ACTION A_LeftTopMove:
IF LeftTopMove THEN
LeftTopBusy:=TRUE;
LeftTopDone:=FALSE;
fb_ton_debug_1(PT:=t#10s);
(*×îºóÔÙ¼ì²éÒ»±éñîºÏ£¬²»ñîºÏÎªÕýÈ·×´Ì¬*)
IF LeftTopLin.NcToPlc.CoupleState<>0 OR LeftBottomLin.NcToPlc.CoupleState<>0
			OR RightTopLin.NcToPlc.CoupleState<>0 OR RightBottomLin.NcToPlc.CoupleState<>0 THEN
			ErrorID:=1;
			LeftTopState:=-100;
END_IF
A_MoveMC();
CASE LeftTopState OF
	0:
		IF Top_MC_MoveAbsolute.Error OR Bottom_MC_MoveAbsolute.Error
			OR RightTopLin_MC_MoveAbsolute.Error OR RightBottomLin_MC_MoveAbsolute.Error THEN		(*¼ì²éMC Error*)
			ErrorID:=2;
			LeftTopState:=99;
		ELSIF leftTopLin.Status.NotMoving AND  leftBottomLin.Status.NotMoving
			 AND RightTopLin.Status.NotMoving AND RightBottomLin.Status.NotMoving THEN	(*Öá¶¼´¦ÓÚÍ£Ö¹×´Ì¬Ê±£¬×ªÏÂÒ»²½*)
			LeftTopState:=1;
		END_IF
	1:
		Top_MC_MoveAbsolute.Position:=LeftTopPosition;
		Top_MC_MoveAbsolute.Velocity:=LeftTopVelocity;
		Top_MC_MoveAbsolute.Execute:=TRUE;
		fb_ton_debug_1.IN:=TRUE;
		LeftTopState:=2;
	2:
		IF RightTopLin.Status.Moving OR LeftBottomLin.Status.Moving OR RightBottomLin.Status.Moving THEN	(*³ýÁËÔË¶¯Öá¶¯£¬ÆäÓàÖáÓÐ¶¯£¬´íÎó*)
			ErrorID:=3;
			LeftTopState:=-100;
		ELSIF NOT Top_MC_MoveAbsolute.Done THEN		(*ÔË¶¯ÖÐ£¬¼ì²éDoneÐÅºÅ£¬Ã»ÓÐÔòÑ­»·£¬³¬Ê±±¨´í*)
			(*IF NOT  fb_ton.Q THEN
				LeftTopState:=2;
			ELSE
				ErrorID:=5;
				LeftTopState:=-100;
			END_IF*)
			LeftTopState:=2;
		ELSIF Top_MC_MoveAbsolute.Done THEN		(*ÔË¶¯Íê³É£¬×ªÏÂÒ»²½*)
				LeftTopState:=88;
		END_IF
		(*½ÓÊÕµ½stopÐÅºÅÊ±£¬reset×´Ì¬*)
		IF LeftTopReset THEN
			LeftTopState:=89;
		END_IF

	88:
		LeftTopMove:=FALSE;
		LeftTopState:=0;
		LeftTopBusy:=FALSE;
		LeftTopDone:=TRUE;
		Error:=FALSE;
		ErrorID:=0;
		Top_MC_MoveAbsolute.Execute:=FALSE;
		fb_ton_debug_1.IN:=FALSE;
	89:
		LeftTopMove:=FALSE;
		LeftTopState:=0;
		LeftTopBusy:=FALSE;
		LeftTopDone:=FALSE;
		Error:=FALSE;
		ErrorID:=0;
		Top_MC_MoveAbsolute.Execute:=FALSE;
		fb_ton_debug_1.IN:=FALSE;
	99:
		LeftTopMove:=FALSE;
		LeftTopState:=99;
		LeftTopBusy:=FALSE;
		LeftTopDone:=FALSE;
		Error:=TRUE;
		Top_MC_MoveAbsolute.Execute:=FALSE;
		fb_ton_debug_1.IN:=FALSE;
	-100:
		FB_PlcEmergencyStop();
		LeftTopMove:=FALSE;
		LeftTopState:=-100;
		LeftTopBusy:=FALSE;
		LeftTopDone:=FALSE;
		Error:=TRUE;
		Top_MC_MoveAbsolute.Execute:=FALSE;
		fb_ton_debug_1.IN:=FALSE;
END_CASE
END_IF
END_ACTION

ACTION A_MoveMC:
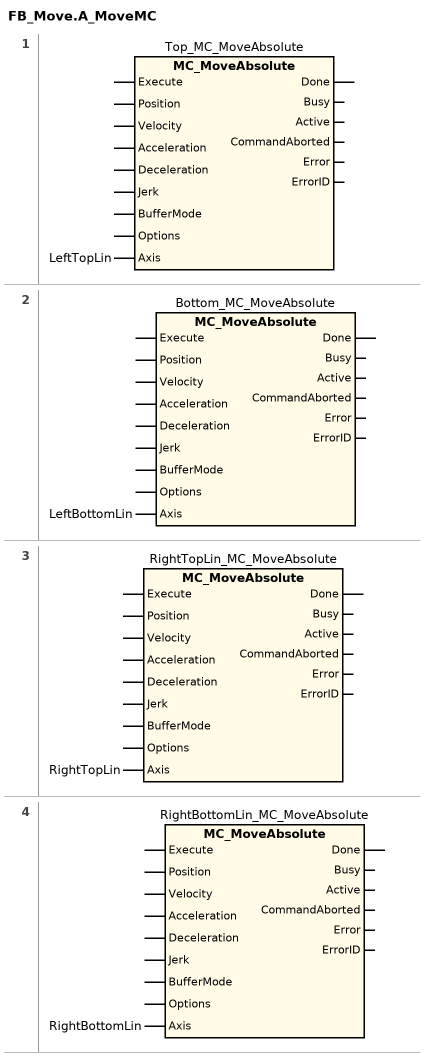
// NETWORK 1
Top_MC_MoveAbsolute(Axis := LeftTopLin); // MC_MoveAbsolute

// NETWORK 2
Bottom_MC_MoveAbsolute(Axis := LeftBottomLin); // MC_MoveAbsolute

// NETWORK 3
RightTopLin_MC_MoveAbsolute(Axis := RightTopLin); // MC_MoveAbsolute

// NETWORK 4
RightBottomLin_MC_MoveAbsolute(Axis := RightBottomLin); // MC_MoveAbsolute
END_ACTION

ACTION A_RightBottomMove:
IF RightBottomMove THEN
RightBottomBusy:=TRUE;
RightBottomDone:=FALSE;
fb_ton_debug_4(PT:=t#10s);
(*×îºóÔÙ¼ì²éÒ»±éñîºÏ£¬²»ñîºÏÎªÕýÈ·×´Ì¬*)
IF LeftTopLin.NcToPlc.CoupleState<>0 OR LeftBottomLin.NcToPlc.CoupleState<>0
			OR RightTopLin.NcToPlc.CoupleState<>0 OR RightBottomLin.NcToPlc.CoupleState<>0 THEN
			ErrorID:=1;
			RightBottomState:=-100;
END_IF
A_MoveMC();
CASE RightBottomState OF
	0:
		IF Top_MC_MoveAbsolute.Error OR Bottom_MC_MoveAbsolute.Error
			OR RightTopLin_MC_MoveAbsolute.Error OR RightBottomLin_MC_MoveAbsolute.Error THEN		(*¼ì²éMC Error*)
			ErrorID:=2;
			RightBottomState:=99;
		ELSIF leftTopLin.Status.NotMoving AND  leftBottomLin.Status.NotMoving
			 AND RightTopLin.Status.NotMoving AND RightBottomLin.Status.NotMoving THEN	(*Öá¶¼´¦ÓÚÍ£Ö¹×´Ì¬Ê±£¬×ªÏÂÒ»²½*)
			RightBottomState:=1;
		END_IF
	1:
		RightBottomLin_MC_MoveAbsolute.Position:=RightBottomPosition;
		RightBottomLin_MC_MoveAbsolute.Velocity:=RightBottomVelocity;
		RightBottomLin_MC_MoveAbsolute.Execute:=TRUE;
		fb_ton_debug_4.IN:=TRUE;
		RightBottomState:=2;
	2:
		IF LeftTopLin.Status.Moving OR RightTopLin.Status.Moving  OR LeftBottomLin.Status.Moving THEN	(*³ýÁËÔË¶¯Öá¶¯£¬ÆäÓàÖáÓÐ¶¯£¬´íÎó*)
			ErrorID:=3;
			RightBottomState:=-100;
		ELSIF NOT RightBottomLin_MC_MoveAbsolute.Done THEN		(*ÔË¶¯ÖÐ£¬¼ì²éDoneÐÅºÅ£¬Ã»ÓÐÔòÑ­»·£¬³¬Ê±±¨´í*)
			(*IF NOT  fb_ton.Q THEN
				LeftTopState:=2;
			ELSE
				ErrorID:=5;
				LeftTopState:=-100;
			END_IF*)
			RightBottomState:=2;
		ELSIF RightBottomLin_MC_MoveAbsolute.Done THEN		(*ÔË¶¯Íê³É£¬×ªÏÂÒ»²½*)
				RightBottomState:=88;
		END_IF
		(*½ÓÊÕµ½stopÐÅºÅÊ±£¬reset×´Ì¬*)
		IF RightBottomReset THEN
			RightBottomState:=89;
		END_IF

	88:
		RightBottomMove:=FALSE;
		RightBottomState:=0;
		RightBottomBusy:=FALSE;
		RightBottomDone:=TRUE;
		Error:=FALSE;
		ErrorID:=0;
		RightBottomLin_MC_MoveAbsolute.Execute:=FALSE;
		fb_ton_debug_4.IN:=FALSE;
	89:
		RightBottomMove:=FALSE;
		RightBottomState:=0;
		RightBottomBusy:=FALSE;
		RightBottomDone:=FALSE;
		Error:=FALSE;
		ErrorID:=0;
		RightBottomLin_MC_MoveAbsolute.Execute:=FALSE;
		fb_ton_debug_4.IN:=FALSE;
	99:
		RightBottomMove:=FALSE;
		RightBottomState:=99;
		RightBottomBusy:=FALSE;
		RightBottomDone:=FALSE;
		Error:=TRUE;
		RightBottomLin_MC_MoveAbsolute.Execute:=FALSE;
		fb_ton_debug_4.IN:=FALSE;
	-100:
		FB_PlcEmergencyStop();
		RightBottomMove:=FALSE;
		RightBottomState:=-100;
		RightBottomBusy:=FALSE;
		RightBottomDone:=FALSE;
		Error:=TRUE;
		RightBottomLin_MC_MoveAbsolute.Execute:=FALSE;
		fb_ton_debug_4.IN:=FALSE;
END_CASE
END_IF
END_ACTION

ACTION A_RightTopMove:
IF RightTopMove THEN
RightTopBusy:=TRUE;
RightTopDone:=FALSE;
fb_ton_debug_2(PT:=t#10s);
(*×îºóÔÙ¼ì²éÒ»±éñîºÏ£¬²»ñîºÏÎªÕýÈ·×´Ì¬*)
IF LeftTopLin.NcToPlc.CoupleState<>0 OR LeftBottomLin.NcToPlc.CoupleState<>0
			OR RightTopLin.NcToPlc.CoupleState<>0 OR RightBottomLin.NcToPlc.CoupleState<>0 THEN
			ErrorID:=1;
			RightTopState:=-100;
END_IF
A_MoveMC();
CASE RightTopState OF
	0:
		IF Top_MC_MoveAbsolute.Error OR Bottom_MC_MoveAbsolute.Error
			OR RightTopLin_MC_MoveAbsolute.Error OR RightBottomLin_MC_MoveAbsolute.Error THEN		(*¼ì²éMC Error*)
			ErrorID:=2;
			RightTopState:=99;
		ELSIF leftTopLin.Status.NotMoving AND  leftBottomLin.Status.NotMoving
			 AND RightTopLin.Status.NotMoving AND RightBottomLin.Status.NotMoving THEN	(*Öá¶¼´¦ÓÚÍ£Ö¹×´Ì¬Ê±£¬×ªÏÂÒ»²½*)
			RightTopState:=1;
		END_IF
	1:
		RightTopLin_MC_MoveAbsolute.Position:=RightTopPosition;
		RightTopLin_MC_MoveAbsolute.Velocity:=RightTopVelocity;
		RightTopLin_MC_MoveAbsolute.Execute:=TRUE;
		fb_ton_debug_2.IN:=TRUE;
		RightTopState:=2;
	2:
		IF LeftTopLin.Status.Moving OR LeftBottomLin.Status.Moving OR RightBottomLin.Status.Moving THEN	(*³ýÁËÔË¶¯Öá¶¯£¬ÆäÓàÖáÓÐ¶¯£¬´íÎó*)
			ErrorID:=3;
			RightTopState:=-100;
		ELSIF NOT RightTopLin_MC_MoveAbsolute.Done THEN		(*ÔË¶¯ÖÐ£¬¼ì²éDoneÐÅºÅ£¬Ã»ÓÐÔòÑ­»·£¬³¬Ê±±¨´í*)
			(*IF NOT  fb_ton.Q THEN
				LeftTopState:=2;
			ELSE
				ErrorID:=5;
				LeftTopState:=-100;
			END_IF*)
			RightTopState:=2;
		ELSIF RightTopLin_MC_MoveAbsolute.Done THEN		(*ÔË¶¯Íê³É£¬×ªÏÂÒ»²½*)
				RightTopState:=88;
		END_IF
		(*½ÓÊÕµ½stopÐÅºÅÊ±£¬reset×´Ì¬*)
		IF RightTopReset THEN
			RightTopState:=89;
		END_IF

	88:
		RightTopMove:=FALSE;
		RightTopState:=0;
		RightTopBusy:=FALSE;
		RightTopDone:=TRUE;
		Error:=FALSE;
		ErrorID:=0;
		RightTopLin_MC_MoveAbsolute.Execute:=FALSE;
		fb_ton_debug_2.IN:=FALSE;
	89:
		RightTopMove:=FALSE;
		RightTopState:=0;
		RightTopBusy:=FALSE;
		RightTopDone:=FALSE;
		Error:=FALSE;
		ErrorID:=0;
		RightTopLin_MC_MoveAbsolute.Execute:=FALSE;
		fb_ton_debug_2.IN:=FALSE;
	99:
		RightTopMove:=FALSE;
		RightTopState:=99;
		RightTopBusy:=FALSE;
		RightTopDone:=FALSE;
		Error:=TRUE;
		RightTopLin_MC_MoveAbsolute.Execute:=FALSE;
		fb_ton_debug_2.IN:=FALSE;
	-100:
		FB_PlcEmergencyStop();
		RightTopMove:=FALSE;
		RightTopState:=-100;
		RightTopBusy:=FALSE;
		RightTopDone:=FALSE;
		Error:=TRUE;
		RightTopLin_MC_MoveAbsolute.Execute:=FALSE;
		fb_ton_debug_2.IN:=FALSE;
END_CASE
END_IF
END_ACTION

ACTION A_TaperMove:
IF TaperMove THEN
TaperBusy:=TRUE;
TaperDone:=FALSE;
fb_ton(PT:=t#80s);
(*×îºóÔÙ¼ì²éÒ»±éñîºÏ£¬²»ñîºÏÎªÕýÈ·×´Ì¬*)
IF LeftTopLin.NcToPlc.CoupleState<>0 OR LeftBottomLin.NcToPlc.CoupleState<>0
			OR RightTopLin.NcToPlc.CoupleState<>0 OR RightBottomLin.NcToPlc.CoupleState<>0 THEN
			ErrorID:=1;
			TaperState:=-100;
END_IF
(*×ó²àÉÏÏÂÖá¶¯£¬ESTOP*)
IF LeftTopLin.Status.Moving OR LeftBottomLin.Status.Moving THEN
			ErrorID:=2;
			TaperState:=-100;
END_IF
(*ÓÒÉÏ¶¯¡¢ÓÒÏÂ²»¶¯£¬»òÕßÓÒÏÂ¶¯¡¢ÓÒÉÏ²»¶¯¡£ESTOP*)
IF (RightTopLin.Status.Moving AND RightBottomLin.Status.NotMoving) OR (RightTopLin.Status.NotMoving AND RightBottomLin.Status.Moving) THEN
			ErrorID:=3;
			TaperState:=-100;
END_IF
A_MoveMC();
CASE TaperState OF

	0:
		IF RightTopLin.Status.Moving OR RightBottomLin.Status.Moving THEN	(*ÓÒ²àÉÏÏÂÖáÕýÔÚÔËÐÐ£¬Ñ­»·¸Ã²½µÈ´ý*)
			TaperState:=88;
		ELSIF Top_MC_MoveAbsolute.Error OR Bottom_MC_MoveAbsolute.Error THEN		(*¼ì²éMC Error*)
			ErrorID:=4;
			TaperState:=99;
		ELSIF leftTopLin.Status.NotMoving AND  leftBottomLin.Status.NotMoving
			 AND RightTopLin.Status.NotMoving AND RightBottomLin.Status.NotMoving THEN	(*Öá¶¼´¦ÓÚÍ£Ö¹×´Ì¬Ê±£¬×ªÏÂÒ»²½*)
			TaperState:=1;
		END_IF
	1:
		RightTopLin_MC_MoveAbsolute.Position:=TaperPosition;
		RightTopLin_MC_MoveAbsolute.Velocity:=TaperVelocity;
		RightBottomLin_MC_MoveAbsolute.Position:=TaperPosition;
		RightBottomLin_MC_MoveAbsolute.Velocity:=TaperVelocity;
		RightTopLin_MC_MoveAbsolute.Execute:=TRUE;
		RightBottomLin_MC_MoveAbsolute.Execute:=TRUE;
		fb_ton.IN:=TRUE;
		TaperState:=2;
	2:
		IF leftTopLin.Status.Moving OR   leftBottomLin.Status.Moving THEN		(*×ó²àÉÏÏÂÖá¶¯£¬ESTOP*)
			ErrorID:=5;
			TaperState:=-100;
		ELSIF  (RightTopLin.Status.Moving AND RightBottomLin.Status.NotMoving) OR (RightTopLin.Status.NotMoving AND RightBottomLin.Status.Moving) THEN
			ErrorID:=6;
			TaperState:=-100;
		ELSIF NOT RightTopLin_MC_MoveAbsolute.Done OR NOT  RightBottomLin_MC_MoveAbsolute.Done THEN		(*ÔË¶¯ÖÐ£¬¼ì²éDoneÐÅºÅ£¬Ã»ÓÐÔòÑ­»·£¬³¬Ê±±¨´í*)
			(*IF NOT  fb_ton.Q THEN
				TaperState:=2;
			ELSE
				ErrorID:=5;
				TaperState:=-100;
			END_IF*)
			TaperState:=2;
		ELSIF RightTopLin_MC_MoveAbsolute.Done  AND  RightBottomLin_MC_MoveAbsolute.Done THEN		(*ÔË¶¯Íê³É£¬×ªÏÂÒ»²½*)
				TaperState:=88;
		END_IF
		(*½ÓÊÕµ½stopÐÅºÅÊ±£¬reset×´Ì¬*)
		IF TaperReset THEN
			TaperState:=89;
		END_IF

	88:
		TaperMove:=FALSE;
		TaperState:=0;
		TaperBusy:=FALSE;
		TaperDone:=TRUE;
		Error:=FALSE;
		ErrorID:=0;
		RightTopLin_MC_MoveAbsolute.Execute:=FALSE;
		RightBottomLin_MC_MoveAbsolute.Execute:=FALSE;
		fb_ton.IN:=FALSE;
	89:
		TaperMove:=FALSE;
		TaperState:=0;
		TaperBusy:=FALSE;
		TaperDone:=FALSE;
		Error:=FALSE;
		ErrorID:=0;
		RightTopLin_MC_MoveAbsolute.Execute:=FALSE;
		RightBottomLin_MC_MoveAbsolute.Execute:=FALSE;
		fb_ton.IN:=FALSE;
	99:
		TaperMove:=FALSE;
		TaperState:=99;
		TaperBusy:=FALSE;
		TaperDone:=FALSE;
		Error:=TRUE;
		RightTopLin_MC_MoveAbsolute.Execute:=FALSE;
		RightBottomLin_MC_MoveAbsolute.Execute:=FALSE;
		fb_ton.IN:=FALSE;
	-100:
		FB_PlcEmergencyStop();
		TaperMove:=FALSE;
		TaperState:=-100;
		TaperBusy:=FALSE;
		TaperDone:=FALSE;
		Error:=TRUE;
		RightTopLin_MC_MoveAbsolute.Execute:=FALSE;
		RightBottomLin_MC_MoveAbsolute.Execute:=FALSE;
		fb_ton.IN:=FALSE;
END_CASE
END_IF
END_ACTION

ACTION A_TopMove:
IF TopMove THEN
TopBusy:=TRUE;
TopDone:=FALSE;
fb_ton1(PT:=t#80s);(*2mm/s max spees,120mmÐÐ³Ì£¬60sÄÚ×ßÍê*)
A_MoveMC();
CASE TopState OF
	0:
		IF Top_MC_MoveAbsolute.Error OR RightTopLin_MC_MoveAbsolute.Error THEN		(*¼ì²éMC Error*)
			ErrorID:=2;
			TopState:=99;
		END_IF
		TopState:=1;
	1:
		Top_MC_MoveAbsolute.Position:=TopPosition;
		Top_MC_MoveAbsolute.Velocity:=TopVelocity;
		Top_MC_MoveAbsolute.Execute:=TRUE;
		RightTopLin_MC_MoveAbsolute.Position:=TopPosition;
		RightTopLin_MC_MoveAbsolute.Velocity:=TopVelocity;
		RightTopLin_MC_MoveAbsolute.Execute:=TRUE;
		fb_ton1.IN:=TRUE;
		TopState:=2;
	2:
		IF leftBottomLin.Status.Moving OR RightBottomLin.Status.Moving THEN	(*ÏÂÁº¶¯,ESTOP*)
			ErrorID:=3;
			TopState:=-100;
		ELSIF  (LeftTopLin.Status.Moving AND  RightTopLin.Status.NotMoving)
				OR (RightTopLin.Status.Moving AND  LeftTopLin.Status.NotMoving) THEN			(*Ò»Öá¶¯£¬ÁíÒ»Öá²»¶¯£¬½ô¼±×´Ì¬*)
			ErrorID:=4;
			TopState:=-100;
		ELSIF NOT Top_MC_MoveAbsolute.Done OR NOT RightTopLin_MC_MoveAbsolute.Done THEN		(*ÔË¶¯ÖÐ£¬¼ì²éDoneÐÅºÅ£¬Ã»ÓÐÔòÑ­»·£¬³¬Ê±±¨´í*)
			TopState:=2;
		ELSIF Top_MC_MoveAbsolute.Done AND RightTopLin_MC_MoveAbsolute.Done THEN		(*ÔË¶¯Íê³É£¬×ªÏÂÒ»²½*)
				TopState:=88;
		END_IF
		(*½ÓÊÕµ½stopÐÅºÅÊ±£¬reset×´Ì¬*)
		IF TopReset THEN
			TopState:=89;
		END_IF

	88:
		TopMove:=FALSE;
		TopState:=0;
		TopBusy:=FALSE;
		TopDone:=TRUE;
		Error:=FALSE;
		ErrorID:=0;
		Top_MC_MoveAbsolute.Execute:=FALSE;
		RightTopLin_MC_MoveAbsolute.Execute:=FALSE;
		fb_ton1.IN:=FALSE;
	89:
		TopMove:=FALSE;
		TopState:=0;
		TopBusy:=FALSE;
		TopDone:=FALSE;
		Error:=FALSE;
		ErrorID:=0;
		Top_MC_MoveAbsolute.Execute:=FALSE;
		RightTopLin_MC_MoveAbsolute.Execute:=FALSE;
		fb_ton1.IN:=FALSE;
	99:
		TopMove:=FALSE;
		TopState:=99;
		TopBusy:=FALSE;
		TopDone:=FALSE;
		Error:=TRUE;
		Top_MC_MoveAbsolute.Execute:=FALSE;
		RightTopLin_MC_MoveAbsolute.Execute:=FALSE;
		fb_ton1.IN:=FALSE;
	-100:
		FB_PlcEmergencyStop();
		TopMove:=FALSE;
		TopState:=-100;
		TopBusy:=FALSE;
		TopDone:=FALSE;
		Error:=TRUE;
		Top_MC_MoveAbsolute.Execute:=FALSE;
		RightTopLin_MC_MoveAbsolute.Execute:=FALSE;
		fb_ton1.IN:=FALSE;
END_CASE
END_IF
END_ACTION

END_FUNCTION_BLOCK

// ---- POUs/CommonFB/MainFB/FB_Stop.TcPOU
FUNCTION_BLOCK FB_Stop
VAR_INPUT
(*È«¾Ö*)
	Mode:DINT;
	PowerState:BOOL;
	CoupleState:DINT;
	(*GapMode*)
	GapStop:BOOL;
	(*BCGapMode*)
	BCGapStop:BOOL;
	(*SingleCarrierMode*)
	TopStop:BOOL;
	BottomStop:BOOL;
	(*TaperMode*)
	TaperStop:BOOL;
	(*DebugMode*)
	LeftTopStop:BOOL;
	RightTopStop:BOOL;
	LeftBottomStop:BOOL;
	RightBottomStop:BOOL;
END_VAR
VAR_OUTPUT
	FbID:DINT:=1001;
	GapState:DINT;
	GapBusy:BOOL;
	GapDone:BOOL;

	BCGapState:DINT;
	BCGapBusy:BOOL;
	BCGapDone:BOOL;

	TopState:DINT;
	TopBusy:BOOL;
	TopDone:BOOL;
	BottomState:DINT;
	BottomBusy:BOOL;
	BottomDone:BOOL;

	TaperState:DINT;
	TaperBusy:BOOL;
	TaperDone:BOOL;

	LeftTopState:DINT;
	LeftTopBusy:BOOL;
	LeftTopDone:BOOL;
	RightTopState:DINT;
	RightTopBusy:BOOL;
	RightTopDone:BOOL;
	LeftBottomState:DINT;
	LeftBottomBusy:BOOL;
	LeftBottomDone:BOOL;
	RightBottomState:DINT;
	RightBottomBusy:BOOL;
	RightBottomDone:BOOL;

	Error:BOOL;
	ErrorID:DINT;
END_VAR
VAR
	Top_MC_Stop: MC_Stop;
	Bottom_MC_Stop: MC_Stop;
	RightTopLin_MC_Stop: MC_Stop;
	RightBottomLin_MC_Stop: MC_Stop;
	fb_ton: TON;
	fb_ton1: TON;
	fb_ton2: TON;
	fb_ton_debug_1:TON;
	fb_ton_debug_2:TON;
	fb_ton_debug_3:TON;
	fb_ton_debug_4:TON;
	fb_ton_BC: TON;
END_VAR

IF PowerState=1 THEN
	IF Mode=1 AND CoupleState=1 THEN
		A_GapStop();
	ELSIF Mode=2 AND CoupleState=0 AND TopStop THEN
		A_TopStop();
	ELSIF Mode=2 AND CoupleState=0 AND BottomStop THEN
		A_BottomStop();
	ELSIF Mode=3 AND CoupleState=0 AND TaperStop THEN
		A_TaperStop();
	ELSIF Mode=4 AND CoupleState=0 AND LeftTopStop THEN
		A_LeftTopStop();
	ELSIF Mode=4 AND CoupleState=0 AND RightTopStop THEN
		A_RightTopStop();
	ELSIF Mode=4 AND CoupleState=0 AND LeftBottomStop THEN
		A_LeftBottomStop();
	ELSIF Mode=4 AND CoupleState=0 AND RightBottomStop THEN
		A_RightBottomStop();
	ELSIF Mode=5 AND CoupleState=0 AND BCGapStop THEN
		A_BCGapStop();
	ELSE
		FB_PlcEmergencyStop();
	END_IF
END_IF

ACTION A_BCGapStop:
IF BCGapStop THEN
BCGapBusy:=TRUE;
BCGapDone:=FALSE;
fb_ton_BC(PT:=t#100ms);
A_StopMC();
CASE BCGapState OF
	0:
		IF Top_MC_Stop.Error OR Bottom_MC_Stop.Error OR RightTopLin_MC_Stop.Error OR RightBottomLin_MC_Stop.Error THEN
			ErrorID:=1;
			BCGapState:=-100;
			Top_MC_Stop.Execute:=FALSE;
			Bottom_MC_Stop.Execute:=FALSE;
			RightTopLin_MC_Stop.Execute:=FALSE;
			RightBottomLin_MC_Stop.Execute:=FALSE;
			A_StopMC();
		ELSE
			BCGapState:=1;
		END_IF
	1:
		Top_MC_Stop.Execute:=TRUE;
		Bottom_MC_Stop.Execute:=TRUE;
		RightTopLin_MC_Stop.Execute:=TRUE;
		RightBottomLin_MC_Stop.Execute:=TRUE;
		fb_ton_BC.IN:=TRUE;
		BCGapState:=2;
	2:
		IF  NOT Top_MC_Stop.Done OR NOT Bottom_MC_Stop.Done OR NOT RightTopLin_MC_Stop.Done OR NOT RightBottomLin_MC_Stop.Done THEN
				BCGapState:=2;
		ELSE
			BCGapState:=88;
			Top_MC_Stop.Execute:=FALSE;
			Bottom_MC_Stop.Execute:=FALSE;
			RightTopLin_MC_Stop.Execute:=FALSE;
			RightBottomLin_MC_Stop.Execute:=FALSE;
			A_StopMC();
		END_IF

	88:
		BCGapStop:=FALSE;
		BCGapState:=0;
		BCGapBusy:=FALSE;
		BCGapDone:=TRUE;
		Error:=FALSE;
		ErrorID:=0;
		fb_ton_BC.IN:=FALSE;

	-100:
		FB_PlcEmergencyStop();
		BCGapStop:=FALSE;
		BCGapState:=-100;
		BCGapBusy:=FALSE;
		BCGapDone:=FALSE;
		Error:=TRUE;
		Top_MC_Stop.Execute:=FALSE;
		Bottom_MC_Stop.Execute:=FALSE;
		RightTopLin_MC_Stop.Execute:=FALSE;
		RightBottomLin_MC_Stop.Execute:=FALSE;
		A_StopMC();
		fb_ton_BC.IN:=FALSE;

END_CASE
END_IF
END_ACTION

ACTION A_BottomStop:
IF BottomStop THEN
BottomBusy:=TRUE;
BottomDone:=FALSE;
fb_ton2(PT:=t#100ms);
A_StopMC();
CASE BottomState OF
	0:
		IF Bottom_MC_Stop.Error OR RightBottomLin_MC_Stop.Error THEN
			ErrorID:=1;
			BottomState:=-100;
			Bottom_MC_Stop.Execute:=FALSE;
			RightBottomLin_MC_Stop.Execute:=FALSE;
			A_StopMC();
		ELSE
			BottomState:=1;
		END_IF
	1:
		Bottom_MC_Stop.Execute:=TRUE;
		RightBottomLin_MC_Stop.Execute:=TRUE;
		fb_ton2.IN:=TRUE;
		BottomState:=2;
	2:
		IF  NOT Bottom_MC_Stop.Done OR NOT Bottom_MC_Stop.Done THEN
				BottomState:=2;
		ELSE
			BottomState:=88;
			Bottom_MC_Stop.Execute:=FALSE;
			RightBottomLin_MC_Stop.Execute:=FALSE;
			A_StopMC();
		END_IF

	88:
		BottomStop:=FALSE;
		BottomState:=0;
		BottomBusy:=FALSE;
		BottomDone:=TRUE;
		Error:=FALSE;
		ErrorID:=0;
		fb_ton2.IN:=FALSE;

	-100:
		FB_PlcEmergencyStop();
		BottomStop:=FALSE;
		BottomState:=-100;
		BottomBusy:=FALSE;
		BottomDone:=FALSE;
		Error:=TRUE;
		Bottom_MC_Stop.Execute:=FALSE;
		RightBottomLin_MC_Stop.Execute:=FALSE;
		A_StopMC();
		fb_ton2.IN:=FALSE;

END_CASE
END_IF
END_ACTION

ACTION A_GapStop:
IF GapStop THEN
GapBusy:=TRUE;
GapDone:=FALSE;
fb_ton(PT:=t#100ms);
A_StopMC();
CASE GapState OF
	0:
		IF Top_MC_Stop.Error OR Bottom_MC_Stop.Error THEN
			ErrorID:=1;
			GapState:=-100;
			Top_MC_Stop.Execute:=FALSE;
			Bottom_MC_Stop.Execute:=FALSE;
			A_StopMC();
		ELSE
			GapState:=1;
		END_IF
	1:
		Top_MC_Stop.Execute:=TRUE;
		Bottom_MC_Stop.Execute:=TRUE;
		fb_ton.IN:=TRUE;
		GapState:=2;
	2:
		IF  NOT Top_MC_Stop.Done OR NOT Bottom_MC_Stop.Done THEN
				GapState:=2;
		ELSE
			GapState:=88;
			Top_MC_Stop.Execute:=FALSE;
			Bottom_MC_Stop.Execute:=FALSE;
			A_StopMC();
		END_IF

	88:
		GapStop:=FALSE;
		GapState:=0;
		GapBusy:=FALSE;
		GapDone:=TRUE;
		Error:=FALSE;
		ErrorID:=0;
		fb_ton.IN:=FALSE;

	-100:
		FB_PlcEmergencyStop();
		GapStop:=FALSE;
		GapState:=-100;
		GapBusy:=FALSE;
		GapDone:=FALSE;
		Error:=TRUE;
		Top_MC_Stop.Execute:=FALSE;
		Bottom_MC_Stop.Execute:=FALSE;
		A_StopMC();
		fb_ton.IN:=FALSE;

END_CASE
END_IF
END_ACTION

ACTION A_LeftBottomStop:
IF LeftBottomStop THEN
LeftBottomBusy:=TRUE;
LeftBottomDone:=FALSE;
fb_ton_debug_3(PT:=t#100ms);
A_StopMC();
CASE LeftBottomState OF
	0:
		IF Bottom_MC_Stop.Error THEN
			ErrorID:=41;
			LeftBottomState:=-100;
			Bottom_MC_Stop.Execute:=FALSE;
			A_StopMC();
		ELSE
			LeftBottomState:=1;
		END_IF
	1:
		Bottom_MC_Stop.Execute:=TRUE;
		fb_ton_debug_3.IN:=TRUE;
		LeftBottomState:=2;
	2:
		IF  NOT Bottom_MC_Stop.Done THEN
				LeftBottomState:=2;
		ELSE
			LeftBottomState:=88;
			Bottom_MC_Stop.Execute:=FALSE;
			A_StopMC();
		END_IF

	88:
		LeftBottomStop:=FALSE;
		LeftBottomState:=0;
		LeftBottomBusy:=FALSE;
		LeftBottomDone:=TRUE;
		Error:=FALSE;
		ErrorID:=0;
		fb_ton_debug_3.IN:=FALSE;

	-100:
		FB_PlcEmergencyStop();
		LeftBottomStop:=FALSE;
		LeftBottomState:=-100;
		LeftBottomBusy:=FALSE;
		LeftBottomDone:=FALSE;
		Error:=TRUE;
		Bottom_MC_Stop.Execute:=FALSE;
		A_StopMC();
		fb_ton_debug_3.IN:=FALSE;

END_CASE
END_IF
END_ACTION

ACTION A_LeftTopStop:
IF LeftTopStop THEN
LeftTopBusy:=TRUE;
LeftTopDone:=FALSE;
fb_ton_debug_1(PT:=t#100ms);
A_StopMC();
CASE LeftTopState OF
	0:
		IF Top_MC_Stop.Error THEN
			ErrorID:=41;
			LeftTopState:=-100;
			Top_MC_Stop.Execute:=FALSE;
			A_StopMC();
		ELSE
			LeftTopState:=1;
		END_IF
	1:
		Top_MC_Stop.Execute:=TRUE;
		fb_ton_debug_1.IN:=TRUE;
		LeftTopState:=2;
	2:
		IF  NOT Top_MC_Stop.Done THEN
				LeftTopState:=2;
		ELSE
			LeftTopState:=88;
			Top_MC_Stop.Execute:=FALSE;
			A_StopMC();
		END_IF

	88:
		LeftTopStop:=FALSE;
		LeftTopState:=0;
		LeftTopBusy:=FALSE;
		LeftTopDone:=TRUE;
		Error:=FALSE;
		ErrorID:=0;
		fb_ton_debug_1.IN:=FALSE;

	-100:
		FB_PlcEmergencyStop();
		LeftTopStop:=FALSE;
		LeftTopState:=-100;
		LeftTopBusy:=FALSE;
		LeftTopDone:=FALSE;
		Error:=TRUE;
		Top_MC_Stop.Execute:=FALSE;
		A_StopMC();
		fb_ton_debug_1.IN:=FALSE;

END_CASE
END_IF
END_ACTION

ACTION A_RightBottomStop:
IF RightBottomStop THEN
RightBottomBusy:=TRUE;
RightBottomDone:=FALSE;
fb_ton_debug_4(PT:=t#100ms);
A_StopMC();
CASE RightBottomState OF
	0:
		IF RightBottomLin_MC_Stop.Error THEN
			ErrorID:=41;
			RightBottomState:=-100;
			RightBottomLin_MC_Stop.Execute:=FALSE;
			A_StopMC();
		ELSE
			RightBottomState:=1;
		END_IF
	1:
		RightBottomLin_MC_Stop.Execute:=TRUE;
		fb_ton_debug_4.IN:=TRUE;
		RightBottomState:=2;
	2:
		IF  NOT RightBottomLin_MC_Stop.Done THEN
				RightBottomState:=2;
		ELSE
			RightBottomState:=88;
			RightBottomLin_MC_Stop.Execute:=FALSE;
			A_StopMC();
		END_IF

	88:
		RightBottomStop:=FALSE;
		RightBottomState:=0;
		RightBottomBusy:=FALSE;
		RightBottomDone:=TRUE;
		Error:=FALSE;
		ErrorID:=0;
		fb_ton_debug_4.IN:=FALSE;

	-100:
		FB_PlcEmergencyStop();
		RightBottomStop:=FALSE;
		RightBottomState:=-100;
		RightBottomBusy:=FALSE;
		RightBottomDone:=FALSE;
		Error:=TRUE;
		RightBottomLin_MC_Stop.Execute:=FALSE;
		A_StopMC();
		fb_ton_debug_4.IN:=FALSE;

END_CASE
END_IF
END_ACTION

ACTION A_RightTopStop:
IF RightTopStop THEN
RightTopBusy:=TRUE;
RightTopDone:=FALSE;
fb_ton_debug_2(PT:=t#100ms);
A_StopMC();
CASE RightTopState OF
	0:
		IF RightTopLin_MC_Stop.Error THEN
			ErrorID:=41;
			RightTopState:=-100;
			RightTopLin_MC_Stop.Execute:=FALSE;
			A_StopMC();
		ELSE
			RightTopState:=1;
		END_IF
	1:
		RightTopLin_MC_Stop.Execute:=TRUE;
		fb_ton_debug_2.IN:=TRUE;
		RightTopState:=2;
	2:
		IF  NOT RightTopLin_MC_Stop.Done THEN
				RightTopState:=2;
		ELSE
			RightTopState:=88;
			RightTopLin_MC_Stop.Execute:=FALSE;
			A_StopMC();
		END_IF

	88:
		RightTopStop:=FALSE;
		RightTopState:=0;
		RightTopBusy:=FALSE;
		RightTopDone:=TRUE;
		Error:=FALSE;
		ErrorID:=0;
		fb_ton_debug_2.IN:=FALSE;

	-100:
		FB_PlcEmergencyStop();
		RightTopStop:=FALSE;
		RightTopState:=-100;
		RightTopBusy:=FALSE;
		RightTopDone:=FALSE;
		Error:=TRUE;
		RightTopLin_MC_Stop.Execute:=FALSE;
		A_StopMC();
		fb_ton_debug_2.IN:=FALSE;

END_CASE
END_IF
END_ACTION

ACTION A_StopMC:
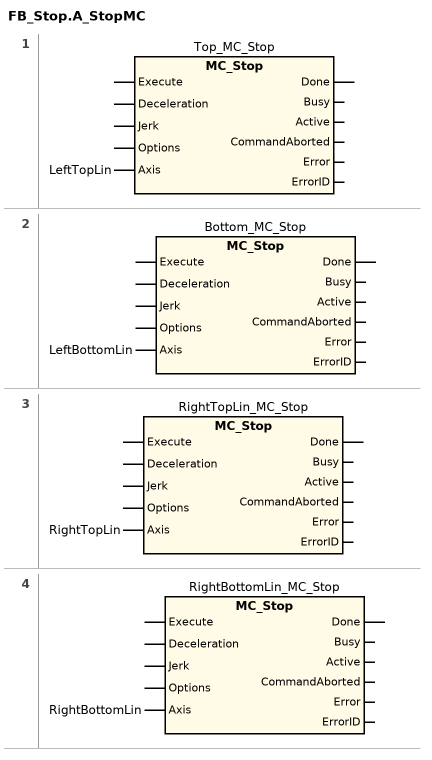
// NETWORK 1
Top_MC_Stop(Axis := LeftTopLin); // MC_Stop

// NETWORK 2
Bottom_MC_Stop(Axis := LeftBottomLin); // MC_Stop

// NETWORK 3
RightTopLin_MC_Stop(Axis := RightTopLin); // MC_Stop

// NETWORK 4
RightBottomLin_MC_Stop(Axis := RightBottomLin); // MC_Stop
END_ACTION

ACTION A_TaperStop:
IF TaperStop THEN
TaperBusy:=TRUE;
TaperDone:=FALSE;
fb_ton(PT:=t#100ms);
A_StopMC();
CASE TaperState OF
	0:
		IF RightTopLin_MC_Stop.Error  OR RightBottomLin_MC_Stop.Error THEN
			ErrorID:=1;
			TaperState:=-100;
			RightTopLin_MC_Stop.Execute:=FALSE;
			RightBottomLin_MC_Stop.Execute:=FALSE;
			A_StopMC();
		ELSE
			TaperState:=1;
		END_IF
	1:
		RightTopLin_MC_Stop.Execute:=TRUE;
		RightBottomLin_MC_Stop.Execute:=TRUE;
		fb_ton.IN:=TRUE;
		TaperState:=2;
	2:
		IF  NOT RightTopLin_MC_Stop.Done OR NOT RightBottomLin_MC_Stop.Done THEN
				TaperState:=2;
		ELSE
			TaperState:=88;
			RightTopLin_MC_Stop.Execute:=FALSE;
			RightBottomLin_MC_Stop.Execute:=FALSE;
			A_StopMC();
		END_IF

	88:
		TaperStop:=FALSE;
		TaperState:=0;
		TaperBusy:=FALSE;
		TaperDone:=TRUE;
		Error:=FALSE;
		ErrorID:=0;
		fb_ton.IN:=FALSE;

	-100:
		FB_PlcEmergencyStop();
		TaperStop:=FALSE;
		TaperState:=-100;
		TaperBusy:=FALSE;
		TaperDone:=FALSE;
		Error:=TRUE;
		RightTopLin_MC_Stop.Execute:=FALSE;
		RightBottomLin_MC_Stop.Execute:=FALSE;
		A_StopMC();
		fb_ton.IN:=FALSE;

END_CASE
END_IF
END_ACTION

ACTION A_TopStop:
IF TopStop THEN
TopBusy:=TRUE;
TopDone:=FALSE;
fb_ton1(PT:=t#100ms);
A_StopMC();
CASE TopState OF
	0:
		IF Top_MC_Stop.Error OR RightTopLin_MC_Stop.Error THEN
			ErrorID:=1;
			TopState:=-100;
			Top_MC_Stop.Execute:=FALSE;
			A_StopMC();
		ELSE
			TopState:=1;
		END_IF
	1:
		Top_MC_Stop.Execute:=TRUE;
		RightTopLin_MC_Stop.Execute:=TRUE;
		fb_ton1.IN:=TRUE;
		TopState:=2;
	2:
		IF  NOT Top_MC_Stop.Done OR NOT RightTopLin_MC_Stop.Done THEN
				TopState:=2;
		ELSE
			TopState:=88;
			Top_MC_Stop.Execute:=FALSE;
			RightTopLin_MC_Stop.Execute:=FALSE;
			A_StopMC();
		END_IF

	88:
		TopStop:=FALSE;
		TopState:=0;
		TopBusy:=FALSE;
		TopDone:=TRUE;
		Error:=FALSE;
		ErrorID:=0;
		fb_ton1.IN:=FALSE;

	-100:
		FB_PlcEmergencyStop();
		TopStop:=FALSE;
		TopState:=-100;
		TopBusy:=FALSE;
		TopDone:=FALSE;
		Error:=TRUE;
		Top_MC_Stop.Execute:=FALSE;
		RightTopLin_MC_Stop.Execute:=FALSE;
		A_StopMC();
		fb_ton1.IN:=FALSE;

END_CASE
END_IF
END_ACTION

END_FUNCTION_BLOCK

// ---- POUs/CommonFB/MainFB/FB_Power.TcPOU
(****************************************************************
NAME:			FB_PowerOn
DATA:			2017.2.16
VERSION:		1.0.0
DESCRIPTION:	FB_PowerOn
HISTORY:
				2017.2.16		NEW

***************************************************************)
FUNCTION_BLOCK FB_Power
VAR_INPUT
	On:BOOL;
	Off:BOOL;
	Check:BOOL;
END_VAR
VAR_OUTPUT
	FbID:DINT:=1001;
	OnState:DINT;
	OffState: INT;
	OnBusy:BOOL;
	OffBusy:BOOL;
	OnStatus:BOOL;
	OffStatus: BOOL;
	Error:BOOL;
	ErrorID:DINT;
	PowerState:BOOL;
END_VAR
VAR
	LeftTopLin_MC_Power: MC_Power;
	RightTopLin_MC_Power: MC_Power;
	LeftBottomLin_MC_Power: MC_Power;
	RightBottomLin_MC_Power: MC_Power;
	fb_ton:TON;
END_VAR

(*power on *)
IF On AND NOT Off THEN
	A_PowerOn();
(*Power Off *)
ELSIF Off AND NOT On THEN
	A_PowerOff();
END_IF
(*Check*)
IF Check THEN
	A_CheckPowerStatus();
END_IF

ACTION A_CheckPowerStatus:
A_PowerMC();
IF  LeftTopLin_MC_Power.Status AND RightTopLin_MC_Power.Status
		AND LeftBottomLin_MC_Power.Status AND RightBottomLin_MC_Power.Status THEN
	PowerState:=1;
ELSIF NOT LeftTopLin_MC_Power.Status AND NOT RightTopLin_MC_Power.Status
		AND NOT LeftBottomLin_MC_Power.Status AND NOT RightBottomLin_MC_Power.Status THEN
	PowerState:=0;
ELSE
	PowerState:=0;
	Error:=TRUE;
	ErrorID:=77;
	(*FB_PlcEmergencyStop();*)
END_IF
END_ACTION

ACTION A_PowerMC:
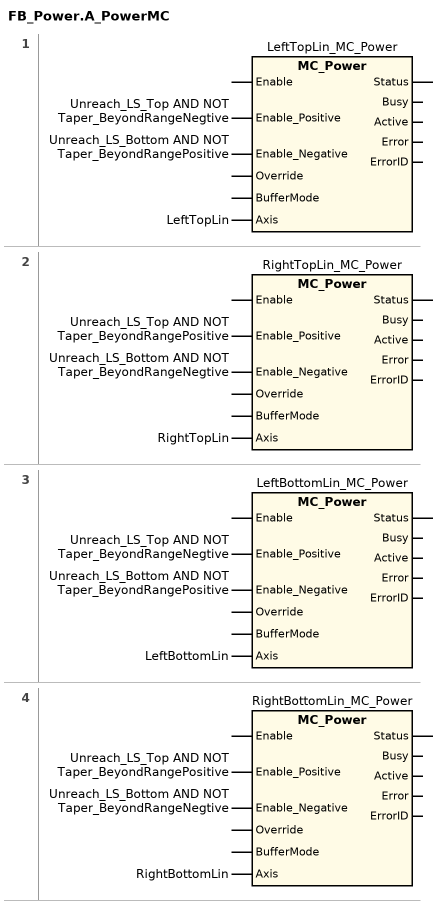
// NETWORK 1
LeftTopLin_MC_Power(
    Enable_Positive := Unreach_LS_Top AND NOT Taper_BeyondRangeNegtive,
    Enable_Negative := Unreach_LS_Bottom AND NOT Taper_BeyondRangePositive,
    Axis := LeftTopLin); // MC_Power

// NETWORK 2
RightTopLin_MC_Power(
    Enable_Positive := Unreach_LS_Top AND NOT Taper_BeyondRangePositive,
    Enable_Negative := Unreach_LS_Bottom AND NOT Taper_BeyondRangeNegtive,
    Axis := RightTopLin); // MC_Power

// NETWORK 3
LeftBottomLin_MC_Power(
    Enable_Positive := Unreach_LS_Top AND NOT Taper_BeyondRangeNegtive,
    Enable_Negative := Unreach_LS_Bottom AND NOT Taper_BeyondRangePositive,
    Axis := LeftBottomLin); // MC_Power

// NETWORK 4
RightBottomLin_MC_Power(
    Enable_Positive := Unreach_LS_Top AND NOT Taper_BeyondRangePositive,
    Enable_Negative := Unreach_LS_Bottom AND NOT Taper_BeyondRangeNegtive,
    Axis := RightBottomLin); // MC_Power
END_ACTION

ACTION A_PowerOff:
(*
IF NOT LeftTopLin_MC_Power.Status OR NOT RightTopLin_MC_Power.Status
			OR NOT LeftBottomLin_MC_Power.Status OR NOT RightBottomLin_MC_Power.Status THEN		(*ÔÙ¼ì²é£¬Öá¶¼Ã»ÓÐPower*)
			LeftTopLin_MC_Power.Enable:=TRUE;
			RightTopLin_MC_Power.Enable:=TRUE;
			LeftBottomLin_MC_Power.Enable:=TRUE;
			RightBottomLin_MC_Power.Enable:=TRUE;
			A_PowerMC();
			fb_ton.IN:=TRUE;
			State:=2;
		ELSE
			ErrorID:=4;
			State:=-100;
		END_IF
*)
OffBusy:=TRUE;
CASE OffState OF
	0:
		IF NOT LeftTopLin_MC_Power.Status AND NOT RightTopLin_MC_Power.Status
			AND NOT LeftBottomLin_MC_Power.Status AND NOT RightBottomLin_MC_Power.Status THEN	(*¶¼Ã»ÉÏµç*)
			OffState:=88;
		ELSE
			OffState:=1;
		END_IF
	1:
		LeftTopLin_MC_Power.Enable:=FALSE;
		RightTopLin_MC_Power.Enable:=FALSE;
		LeftBottomLin_MC_Power.Enable:=FALSE;
		RightBottomLin_MC_Power.Enable:=FALSE;
		A_PowerMC();
		OffState:=2;
	2:
		IF NOT LeftTopLin_MC_Power.Status AND NOT RightTopLin_MC_Power.Status
			AND NOT LeftBottomLin_MC_Power.Status AND NOT RightBottomLin_MC_Power.Status THEN	(*¶¼Ã»ÉÏµç*)
			OffState:=88;
		ELSE
			ErrorId:=11;
			OffState:=-100;
		END_IF
	88:
		Off:=FALSE;
		OffState:=0;
		OffBusy:=FALSE;
		OnStatus:=FALSE;
		OffStatus:=TRUE;
		Error:=FALSE;
		ErrorID:=0;
	-100:
		FB_PlcEmergencyStop();
		Off:=FALSE;
		OffState:=-100;
		OffBusy:=FALSE;
		OffStatus:=FALSE;
		Error:=TRUE;

END_CASE
END_ACTION

ACTION A_PowerOn:
OnBusy:=TRUE;
fb_ton(PT:=t#0.5s);
CASE OnState OF
	0:	(*Check*)
		A_PowerMC();
		IF LeftTopLin_MC_Power.Error OR RightTopLin_MC_Power.Error
			OR LeftBottomLin_MC_Power.Error OR RightBottomLin_MC_Power.Error
			OR NOT LeftTopLin_MC_Power.Active OR NOT RightTopLin_MC_Power.Active
			OR NOT LeftBottomLin_MC_Power.Active OR NOT RightBottomLin_MC_Power.Active THEN		(*FB Error*)
			ErrorID:=1;
			OnState:=99;
		ELSIF LeftTopLin_MC_Power.Status OR RightTopLin_MC_Power.Status
			OR LeftBottomLin_MC_Power.Status OR RightBottomLin_MC_Power.Status THEN		(*ÖáÒÑ¾­¶¼PowerOn£¬²»·ûºÏ¹¦ÄÜ¿éµ÷ÓÃÌõ¼þ*)
			ErrorID:=2;
			OnState:=-100;
		ELSIF NOT LeftTopLin_MC_Power.Status OR NOT RightTopLin_MC_Power.Status
			OR NOT LeftBottomLin_MC_Power.Status OR NOT RightBottomLin_MC_Power.Status THEN		(*Öá¶¼Ã»ÓÐPower£¬×ªÏÂÒ»²½*)
			OnState:=1;
		ELSE
			ErrorID:=3;
			OnState:=-100;
		END_IF
	1:	(*Execute*)
		IF NOT LeftTopLin_MC_Power.Status OR NOT RightTopLin_MC_Power.Status
			OR NOT LeftBottomLin_MC_Power.Status OR NOT RightBottomLin_MC_Power.Status THEN		(*ÔÙ¼ì²é£¬Öá¶¼Ã»ÓÐPower*)
			LeftTopLin_MC_Power.Enable:=TRUE;
			RightTopLin_MC_Power.Enable:=TRUE;
			LeftBottomLin_MC_Power.Enable:=TRUE;
			RightBottomLin_MC_Power.Enable:=TRUE;
			A_PowerMC();
			fb_ton.IN:=TRUE;
			OnState:=2;
		ELSE
			ErrorID:=4;
			OnState:=-100;
		END_IF
	2:	(*Wait*)
		A_PowerMC();
		IF NOT LeftTopLin_MC_Power.Status OR NOT RightTopLin_MC_Power.Status
			OR NOT LeftBottomLin_MC_Power.Status OR NOT RightBottomLin_MC_Power.Status THEN		(*Power StatusÐÅºÅ²»µ½£¬¼ÌÐøµÈ´ý£¬Èç¹û³¬Ê±ÔòFB Error*)
			IF NOT fb_ton.Q THEN
				OnState:=2;
			ELSE
				ErrorID:=8;
				OnState:=99;
			END_IF
		ELSIF  LeftTopLin_MC_Power.Status AND RightTopLin_MC_Power.Status
			AND LeftBottomLin_MC_Power.Status AND RightBottomLin_MC_Power.Status THEN			(*ÕýÈ·µç»úÉÏµã×´Ì¬£¬×ªÏÂÒ»²½*)
				OnState:=88;
		ELSE
				ErrorID:=9;
				OnState:=-100;
		END_IF
	88:
		On:=FALSE;
		OnState:=0;
		OnBusy:=FALSE;
		OnStatus:=TRUE;
		OffStatus:=FALSE;
		Error:=FALSE;
		ErrorID:=0;
		fb_ton.IN:=FALSE;
	99:
		On:=FALSE;
		OnState:=99;
		OnBusy:=FALSE;
		OnStatus:=FALSE;
		Error:=TRUE;
		LeftTopLin_MC_Power.Enable:=FALSE;
		RightTopLin_MC_Power.Enable:=FALSE;
		LeftBottomLin_MC_Power.Enable:=FALSE;
		RightBottomLin_MC_Power.Enable:=FALSE;
		fb_ton.IN:=FALSE;
	-100:
		FB_PlcEmergencyStop();
		On:=FALSE;
		OnState:=-100;
		OnBusy:=FALSE;
		OnStatus:=FALSE;
		Error:=TRUE;
		LeftTopLin_MC_Power.Enable:=FALSE;
		RightTopLin_MC_Power.Enable:=FALSE;
		LeftBottomLin_MC_Power.Enable:=FALSE;
		RightBottomLin_MC_Power.Enable:=FALSE;
		fb_ton.IN:=FALSE;

END_CASE
END_ACTION

END_FUNCTION_BLOCK

// ---- POUs/2.SingleMotorMode/TaperMode/TaperMode.TcPOU
PROGRAM TaperMode
VAR
	(*key Command*)
	btn_PowerOn: BOOL;
	btn_PowerOff: BOOL;
	TaperLargePositionNew:LREAL;
	TaperLargePositionActual: LREAL;
	TaperPositionNew:LREAL;
	TaperVelocityNew:LREAL;
	btn_TaperMove:BOOL;
	btn_TaperStop:BOOL;
	(*Var*)
	fb_ton1:TON;
	fb_ton2:TON;
	(*Status*)
	State:DINT;
	Busy:BOOL;
	InitDone:BOOL;
	Error:BOOL;
	ErrorID:DINT;
	m_state: DINT;
	s_state: DINT;
	ton_t: TON;
	range_state: DINT;
	d_state: DINT;
	(*¼ì²âµ½ÏÞÎ»£¬»Ö¸´Move×´Ì¬*)
	FTrig_ReachLS: F_TRIG;
	FTrig_btn_GapMove: F_TRIG;
	btn_Power: BOOL;
END_VAR

TaperPositionActual:=((Pos_RightTopLin+Pos_RighTBottomLin)-(Pos_LeftTopLin+Pos_LeftBottomLin))/2;	(*Êµ¼ÊTaper¶È£¬Taper¶¨ÒåÎªµ¥²à*)
TaperVelocityActual:=(Velo_RightTopLin+Velo_RightBottomLin)/2;
TaperLargePositionActual:=TaperPositionActual+(Pos_LeftTopLin+Pos_LeftBottomLin)/2;					(*´óTaper=Taper¶È+×ó²àGap*)
TaperLargePositionNew:=TaperPositionNew+(Pos_LeftTopLin+Pos_LeftBottomLin)/2;					(*´óTaper=Taper¶È+×ó²àGap*)
(*********************************************************************Monitor All Carrirt Position***********************************************)
A_MonitoringAllAxis();
(*********************************************************************A_PosDiffDetection***********************************************)
A_PosDiffDetection();
(*********************************************************************btn_PowerOn************************************************************)
IF btn_Power AND st_Power=0 THEN
	btn_PowerOn:=TRUE;
	btn_Power:=FALSE;
END_IF
IF btn_Power AND st_Power=1 THEN
	btn_PowerOff:=TRUE;
	btn_Power:=FALSE;
END_IF
(*********************************************************************btn_PowerOn************************************************************)
IF btn_PowerOn THEN
	A_PowerOn();
END_IF
(******************************************************ÉÏµç×´Ì¬£¬´¦ÓÚñîºÏ×´Ì¬£¬ESTOP***********************************************)
IF NOT btn_PowerOff THEN
	IF st_Power=1 AND st_Couple<>0THEN
		Error:=TRUE;
		ErrorID:=101;
		FB_PlcEmergencyStop();
		LED_Error:=TRUE;
	END_IF
END_IF
(*********************************************************************btn_Move*****************************************************************)
IF InitDone THEN
	IF btn_TaperMove THEN
		CASE m_state OF
			0:
				FB_Move.Mode:=3;						(*1£ºgapÄ£Ê½£»2£ºµ¥ÁºÄ£Ê½£¬3£ºtaperÄ£Ê½*)
				FB_Move.CoupleState:=st_Couple;			(*ñîºÏ×´Ì¬ÊäÈë*)
				FB_Move.PowerState:=st_Power;			(*µçÔ´×´Ì¬ÊäÈë*)
				FB_Move.TaperMove:=TRUE;				(*Execute TRUE*)
				FB_Move.TaperPosition:=TaperLargePositionNew;	(*Î»ÖÃ*)
				FB_Move.TaperVelocity:=TaperVelocityNew;	(*ËÙ¶È*)
				FB_Move();								(*Æô¶¯FB*)
				m_state:=1;
			1:
				FB_Move();
				IF NOT FB_Move.TaperDone THEN			(*ÔË¶¯Î´Íê³É£¬Ñ­»·*)
					m_state:=1;
					LED_Run:=TRUE;
				ELSE									(*ÔË¶¯Íê³É£¬ÏÂÒ»²½*)
					m_state:=88;
				END_IF

			88:
				btn_TaperMove:=FALSE;					(*×´Ì¬»Ö¸´*)
				m_state:=0;
				LED_Run:=FALSE;
		END_CASE
	END_IF
END_IF
(*******************************************************************btn_Stop********************************************************************)
IF btn_TaperStop THEN
	LED_Run:=FALSE;
	TaperMoveIndicator:=0;
	FB_Move.TaperReset:=TRUE;							(*¸øÔË¶¯FB¸øÍ£Ö¹ÐÅºÅ£¬Ê¹FB_Move×´Ì¬»Ö¸´*)
	FB_Move();											(*Æô¶¯FB_Move*)
	btn_TaperMove:=FALSE;								(*btn_GapMove:=FALSE*)
	m_state:=0;											(*m_state:=0;*)
	CASE s_state OF
			0:
				FB_Stop.Mode:=3;							(*1£ºgapÄ£Ê½£»2£ºµ¥ÁºÄ£Ê½£»3£ºtaperÄ£Ê½*)
				FB_Stop.CoupleState:=st_Couple;			(*ñîºÏ×´Ì¬ÊäÈë*)
				FB_Stop.PowerState:=st_Power;				(*µçÔ´×´Ì¬ÊäÈë*)
				FB_Stop.TaperStop:=TRUE;				(*Execute TRUE*)
				FB_Stop();								(*Æô¶¯FB*)
				s_state:=1;
			1:
				FB_Stop();
				IF NOT FB_Stop.TaperDone THEN			(*Í£Ö¹Î´Íê³É£¬Ñ­»·*)
					s_state:=1;
				ELSE									(*Í£Ö¹Íê³É£¬ÏÂÒ»²½*)
					s_state:=88;
				END_IF
			88:
				btn_TaperStop:=FALSE;						(*»Ö¸´×´Ì¬*)
				FB_Move.TaperReset:=FALSE;					(*ÔËÐÐFB*)
				s_state:=0;
		END_CASE

END_IF
(****************************TaperMoveIndicator***************************)
IF TaperVelocityActual>0 THEN
	TaperMoveIndicator:=1;
ELSIF TaperVelocityActual<0 THEN
	TaperMoveIndicator:=-1;
ELSE
	TaperMoveIndicator:=0;
END_IF
(*********************************************************************btn_PowerOff************************************************************)
IF btn_PowerOff THEN
	A_PowerOff();
END_IF
(*********************************************************************ÏÞÎ»Åö´¥×´Ì¬»Ö¸´************************************************************)
(*Èç¹û¼ì²âµ½ÏØÏÞÎ»¿ª¹ØÏÂ½µÑØ£¬»Ö¸´Move×´Ì¬*)
FTrig_ReachLS(CLK:=Unreach_LS_Top AND Unreach_LS_Bottom);
IF FTrig_ReachLS.Q THEN
	btn_TaperStop:=TRUE;
END_IF
(*Èç¹û¼ì²âµ½TopÏÞÎ»¿ª¹ØFALSE£¬ÇÒÄ¿±êÎ»ÖÃ´óÓÚµ±Ç°Î»ÖÃÊ±£¬»òÕßÏà·´Ê±£¬»Ö¸´Move×´Ì¬*)
IF NOT Unreach_LS_Top AND TaperLargePositionNew-TaperLargePositionActual>0.0005 AND btn_TaperMove THEN
	btn_TaperStop:=TRUE;
END_IF
IF NOT Unreach_LS_Bottom AND TaperLargePositionNew-TaperLargePositionActual<0.0005 AND btn_TaperMove THEN
	btn_TaperStop:=TRUE;
END_IF

ACTION A_MonitoringAllAxis:
(****************************************************************
NAME:			A_MonitoringAllAxis
DATA:			2017.3.20
VERSION:		1.0.0
DESCRIPTION:	
				Ã¿´ÎÑ­»·¾ùÖ´ÐÐÖáÎ»ÖÃºÍÖáÔË¶¯µÄ¼ì²é
				1.4ÖáÏà¶ÔÔË¶¯¼ì²é
				2.4Öá¹âÕ¤³ßÎ»ÖÃ¡¢ËÙ¶È¶Ô±È¼ì²é
				3.Ã¿Öá¹âÕ¤ºÍ±àÂëÆ÷Î»ÖÃ¶Ô±È¼ì²é
HISTORY:
				2017.3.27		NEW

***************************************************************)
(*************************************************************************************1.4ÖáÏà¶ÔÔË¶¯¼ì²é************************************************************************************)
(*³ýÁËÓÒÉÏºÍÓÒÏÂÖáÒ»Æð¶¯£¬ÆäÓàÖá¶¯¶¼ESTOP*)
(*×óÉÏ¡¢×óÏÂÖá¶¯*)
IF  LeftTopLin.Status.Moving OR LeftBottomLin.Status.Moving THEN
	btn_TaperStop:=TRUE;
	FB_PlcEmergencyStop();
	Error:=TRUE;
	ErrorID:=11;
	LED_Error:=TRUE;
END_IF
(*ÓÒÉÏ¶¯¡¢ÓÒÏÂ²»¶¯£¬»òÕßÓÒÏÂ¶¯¡¢ÓÒÉÏ²»¶¯¡£ESTOP*)
IF (RightTopLin.Status.Moving AND NOT RightBottomLin.Status.Moving) OR (NOT RightTopLin.Status.Moving AND RightBottomLin.Status.Moving) THEN
	btn_TaperStop:=TRUE;
	FB_PlcEmergencyStop();
	Error:=TRUE;
	ErrorID:=12;
	LED_Error:=TRUE;
END_IF
(*************************************************************************************2.4Öá¹âÕ¤³ßÎ»ÖÃ¡¢ËÙ¶È¶Ô±È¼ì²é**********************************************************************)
IF st_power<>0 THEN
(*Top×óÓÒºÍBottom×óÓÒ Î»ÖÃ±È¶Ô£¬³¬³öRangeÊ±£¬µç»úEnable_Positive=false*)
IF (Pos_RightTopLin-Pos_leftTopLin>Range_TaperPos/2) OR (Pos_RightBottomLin-Pos_leftBottomLin>Range_TaperPos/2) THEN
	Taper_BeyondRangePositive:=TRUE;
ELSE
	Taper_BeyondRangePositive:=FALSE;
END_IF
(*TopÓÒÐ¡ÓÚ×óºÍBottomÓÒÐ¡ÓÚ×ó£¬ Î»ÖÃ±È¶Ô£¬³¬³öDiffÊ±£¬µç»úEnable_Negtive=false*)
IF  (Pos_leftTopLin-Pos_RightTopLin>Threshold_TaperTopPos) OR (Pos_leftBottomLin-Pos_RightBottomLin>Threshold_TaperBottomPos) THEN
	Taper_BeyondRangeNegtive:=TRUE;
ELSE
	Taper_BeyondRangeNegtive:=FALSE;
END_IF
(*×óÖáÉÏÏÂÎ»ÖÃËÙ¶È¶Ô±È£¬³¬³öESTOP*)
IF ABS(Pos_LeftTopLin-Pos_LeftBottomLin)>Threshold_TaperLeftPos  THEN
	btn_TaperStop:=TRUE;
	FB_PlcEmergencyStop();
	Error:=TRUE;
	ErrorID:=13;
	LED_Error:=TRUE;
ELSIF  ABS(Velo_leftTopLin-Velo_LeftBottomLin)>Threshold_TaperLeftVelo THEN
	(*btn_TaperStop:=TRUE;
	FB_PlcEmergencyStop();*)
	Error:=TRUE;
	ErrorID:=14;
END_IF
(*ÓÒÖáÉÏÏÂÎ»ÖÃËÙ¶È¶Ô±È£¬³¬³öESTOP*)
IF ABS(Pos_RightTopLin-Pos_RightBottomLin)>Threshold_TaperRightPos  THEN
	btn_TaperStop:=TRUE;
	FB_PlcEmergencyStop();
	Error:=TRUE;
	ErrorID:=15;
	LED_Error:=TRUE;
ELSIF  ABS(Velo_RightTopLin-Velo_RightBottomLin)>Threshold_TaperRightVelo THEN
	(*btn_TaperStop:=TRUE;
	FB_PlcEmergencyStop();*)
	Error:=TRUE;
	ErrorID:=16;
END_IF
END_IF
(*********************************************************************************3.Ã¿Öá¹âÕ¤ºÍ±àÂëÆ÷Î»ÖÃ¶Ô±È¼ì²é**********************************************************************)
END_ACTION

ACTION A_PosDiffDetection:
IF ABS(PosDiff_LeftTopLin_actual-PosDiff_RightTopLin_actual)>0.2 THEN
	ErrorID:=51;
	Error:=TRUE;
	btn_TaperStop:=TRUE;
	FB_PlcEmergencyStop();
	LED_Error:=TRUE;
ELSIF ABS(PosDiff_LeftBottomLin_actual-PosDiff_RightBottomLin_actual)>0.2 THEN
	ErrorID:=53;
	Error:=TRUE;
	btn_TaperStop:=TRUE;
	FB_PlcEmergencyStop();
	LED_Error:=TRUE;
END_IF
END_ACTION

ACTION A_PowerOff:
CASE d_state OF
		0:(*PowerOff*)
			FB_Power(Off:=TRUE);
				d_state:=1;
		1:
			IF NOT FB_power.OffStatus THEN
				d_state:=1;
			ELSE
				d_state:=88;
			END_IF
		88:(*ResetAllState*)
			btn_PowerOn:=FALSE;
			btn_TaperMove:=FALSE;
			btn_TaperStop:=FALSE;
			fb_ton1.IN:=FALSE;
			fb_ton2.IN:=FALSE;
			ton_t.IN:=FALSE;
			State:=0;
			Busy:=FALSE;
			InitDone:=FALSE;
			Error:=FALSE;
			ErrorID:=0;
			m_state:=0;
			s_state:=0;
			btn_PowerOff:=FALSE;
			d_state:=0;
			LED_Error:=FALSE;
			LED_Run:=FALSE;
END_CASE
END_ACTION

ACTION A_powerOn:
(****************************************************************
NAME:			A_SetAxisPositionAndPowerOn
DATA:			2017.3.27
VERSION:		1.0.0
DESCRIPTION:	
				ÉÏµãÃüÁîºó£¬Ë³ÐòÖ´ÐÐ£º
				1.FB_SetAxisPosition
				2.FB_PowerOn
				·µ»ØÖ´ÐÐÊÇ·ñ³É¹¦
HISTORY:
				2017.3.27		NEW
				2017.5.8		É¾³ýÁËsetAxisPosition£¬ÒÆ¶¯µ½MAIN³ÌÐòÖÐ
							±ä¸üNAMEÎªA_PowerOn

***************************************************************)
fb_ton2(PT:=t#0.5s);
CASE State OF
	0:	(*FB_Power_On*)
		FB_Power(On:=TRUE);
		fb_ton2.IN:=TRUE;
		State:=1;
	1:	(*wait*)
		FB_power();
		IF NOT FB_power.OnStatus THEN		(*FB_Power_OnÃ»ÓÐÖ´ÐÐÍê£¬wait£¬³¬Ê±FB Error*)
			IF NOT fb_ton2.Q THEN
				State:=1;
			ELSE
				ErrorID:=1;
				State:=99;
			END_IF
		ELSE
			State:=88;
		END_IF
	88:	(*All Done*)
		btn_PowerOn:=FALSE;
		State:=0;
		Error:=FALSE;
		ErrorID:=0;
		Busy:=FALSE;
		InitDone:=TRUE;
		FB_power.On:=FALSE;
		fb_ton1.IN:=FALSE;
		fb_ton2.IN:=FALSE;
	99:
		btn_PowerOn:=FALSE;
		State:=99;
		Error:=TRUE;
		Busy:=FALSE;
		InitDone:=FALSE;
		FB_Power.On:=FALSE;
		fb_ton1.IN:=FALSE;
		fb_ton2.IN:=FALSE;
		LED_Error:=TRUE;
END_CASE
END_ACTION

END_PROGRAM

// ---- POUs/1.CarrierMode/GapMode/GapMode.TcPOU
PROGRAM GapMode
VAR
	(*key Command*)
	btn_PowerOn: BOOL;
	btn_PowerOff: BOOL;
	(*GapMode*)
	GapPositionNew:LREAL:=20;
	GapVelocityNew:LREAL:=1;
	btn_GapMove:BOOL;
	btn_GapStop:BOOL;
	(*Var*)
	fb_ton1:TON;
	fb_ton2:TON;
	fb_ton3:TON;
	(*Status*)
	State:DINT;
	Busy:BOOL;
	InitDone:BOOL;
	(*FB*)

	m_state: DINT;
	s_state: DINT;
	(*¼ì²âµ½ÏÞÎ»£¬»Ö¸´Move×´Ì¬*)
	FTrig_ReachLS: F_TRIG;
	FTrig_btn_GapMove: F_TRIG;
	GapOutRange: BOOL;
	(*PowerOff*)
	d_state: DINT;
	LL: LREAL;
	LL2: LREAL;
	BB:LREAL;
	AA:LREAL;
	CC:LREAL;
	DD:LREAL;
	btn_Power: BOOL;
END_VAR

GapPositionActual:=(Pos_LeftTopLin+Pos_LeftBottomLin+Pos_RightTopLIn+Pos_RightBottomLIn)/2;
GapVelocityActual:=(Velo_LeftTopLin+Velo_LeftBottomLin+Velo_RightTopLIn+Velo_RightBottomLIn)/2;
(*********************************************************************btn_PowerOn************************************************************)
IF btn_Power AND st_Power=0 THEN
	btn_PowerOn:=TRUE;
	btn_Power:=FALSE;
END_IF
IF btn_Power AND st_Power=1 THEN
	btn_PowerOff:=TRUE;
	btn_Power:=FALSE;
END_IF
(*********************************************************************btn_PowerOn************************************************************)
IF btn_PowerOn THEN
	A_CoupleAxisAndPowerOn();
END_IF
(******************************************************ÉÏµç×´Ì¬£¬²»´¦ÓÚñîºÏ×´Ì¬£¬ESTOP***********************************************)
IF NOT btn_PowerOff THEN
	IF st_Power=1 AND st_Couple<>1THEN
		Error:=TRUE;
		ErrorID:=101;
		FB_PlcEmergencyStop();
		LED_Error:=TRUE;
	END_IF
END_IF
(*********************************************************************Monitor All Carrirt Position***********************************************)
A_MonitoringAllAxis();
(*********************************************************************A_PosDiffDetection***********************************************)
A_PosDiffDetection();
(*********************************************************************btn_Move*****************************************************************)
IF InitDone THEN
	IF btn_GapMove THEN
		CASE m_state OF
			0:
				FB_Move.Mode:=1;						(*1£ºgapÄ£Ê½£»2£ºµ¥ÁºÄ£Ê½£¬3£ºtaperÄ£Ê½*)
				FB_Move.CoupleState:=st_Couple;			(*ñîºÏ×´Ì¬ÊäÈë*)
				FB_Move.PowerState:=st_Power;			(*µçÔ´×´Ì¬ÊäÈë*)
				FB_Move.GapMove:=TRUE;				(*Execute TRUE*)
				FB_Move.GapPosition:=GapPositionNew;		(*Î»ÖÃ*)
				FB_Move.GapVelocity:=GapVelocityNew;		(*ËÙ¶È*)
				FB_Move();								(*Æô¶¯FB*)
				IF GapPositionNew-GapPositionActual>0.001 THEN	(*ÔË¶¯·½ÏòÖ¸Ê¾*)
					GapMoveIndicator:=1;
				ELSIF GapPositionNew-GapPositionActual<0.001 THEN
					GapMoveIndicator:=-1;
				ELSE
					GapMoveIndicator:=0;
				END_IF
				m_state:=1;
			1:
				FB_Move();
				IF NOT FB_Move.GapDone THEN			(*ÔË¶¯Î´Íê³É£¬Ñ­»·*)
					Led_Run:=TRUE;
					m_state:=1;

				ELSE									(*ÔË¶¯Íê³É£¬ÏÂÒ»²½*)
					m_state:=88;
				END_IF
			88:
				btn_GapMove:=FALSE;					(*×´Ì¬»Ö¸´*)
				Led_Run:=FALSE;
				m_state:=0;
		END_CASE
	END_IF
END_IF
(*******************************************************************btn_Stop********************************************************************)
IF btn_GapStop THEN
	Led_Run:=FALSE;
	GapMoveIndicator:=0;
	FB_Move.GapReset:=TRUE;							(*¸øÔË¶¯FB¸øÍ£Ö¹ÐÅºÅ£¬Ê¹FB_Move×´Ì¬»Ö¸´*)
	FB_Move();											(*Æô¶¯FB_Move*)
	btn_GapMove:=FALSE;								(*btn_GapMove:=FALSE*)
	m_state:=0;											(*m_state:=0;*)
	CASE s_state OF
			0:
				FB_Stop.Mode:=1;							(*1£ºgapÄ£Ê½£»2£ºµ¥ÁºÄ£Ê½£»3£ºtaperÄ£Ê½*)
				FB_Stop.CoupleState:=st_Couple;			(*ñîºÏ×´Ì¬ÊäÈë*)
				FB_Stop.PowerState:=st_Power;				(*µçÔ´×´Ì¬ÊäÈë*)
				FB_Stop.GapStop:=TRUE;					(*Execute TRUE*)
				FB_Stop();								(*Æô¶¯FB*)
				s_state:=1;
			1:
				FB_Stop();
				IF NOT FB_Stop.GapDone THEN			(*Í£Ö¹Î´Íê³É£¬Ñ­»·*)
					s_state:=1;
				ELSE									(*Í£Ö¹Íê³É£¬ÏÂÒ»²½*)
					s_state:=88;
				END_IF
			88:
				btn_GapStop:=FALSE;						(*»Ö¸´×´Ì¬*)
				FB_Move.GapReset:=FALSE;				(*ÔËÐÐFB*)
				s_state:=0;
		END_CASE

END_IF
(*********************************************************************btn_PowerOff************************************************************)
IF btn_PowerOff THEN
	A_DecoupleAndPowerOff();
END_IF
(*********************************************************************ÏÞÎ»Åö´¥×´Ì¬»Ö¸´************************************************************)
(*Èç¹û¼ì²âµ½ÏØÏÞÎ»¿ª¹ØÏÂ½µÑØ£¬»Ö¸´Move×´Ì¬*)
FTrig_ReachLS(CLK:=Unreach_LS_Top AND Unreach_LS_Bottom);
IF FTrig_ReachLS.Q THEN
	btn_GapStop:=TRUE;
END_IF
(*Èç¹û¼ì²âµ½TopÏÞÎ»¿ª¹ØFALSE£¬ÇÒÄ¿±êÎ»ÖÃ´óÓÚµ±Ç°Î»ÖÃÊ±£¬»òÕßÏà·´Ê±£¬»Ö¸´Move×´Ì¬*)
IF NOT Unreach_LS_Top AND GapPositionNew-GapPositionActual>0.0005 AND btn_GapMove THEN
	btn_GapStop:=TRUE;
END_IF
IF NOT Unreach_LS_Bottom AND GapPositionNew-GapPositionActual<0.0005 AND btn_GapMove THEN
	btn_GapStop:=TRUE;
END_IF

ACTION A_CoupleAxisAndPowerOn:
(****************************************************************
NAME:			A_SetAxisPositionAndCoupleAxisAndPowerOn
DATA:			2017.2.16
VERSION:		1.0.0
DESCRIPTION:	
				ÉÏµãÃüÁîºó£¬Ë³ÐòÖ´ÐÐ£º
				1.FB_SetAxisPosition
				2.FB_CoupleAxis
				3.FB_PowerOn
				·µ»ØÖ´ÐÐÊÇ·ñ³É¹¦
HISTORY:
				2017.2.16		NEW

***************************************************************)
fb_ton2(PT:=t#0.5s);
fb_ton3(PT:=t#0.5s);
FB_CoupleAxis();
CASE State OF
	0:	(*FB_Couple_Axis*)
		FB_CoupleAxis(Execute:=TRUE);
		fb_ton2.IN:=TRUE;
		State:=1;
	1:	(*wait*)

		IF NOT FB_CoupleAxis.InGear THEN		(*FB_Couple_AxisÃ»ÓÐÖ´ÐÐÍê£¬wait£¬³¬Ê±FB Error*)
			IF NOT fb_ton1.Q THEN
				State:=1;
			ELSE
				ErrorID:=1;
				State:=99;
			END_IF
		ELSE
			State:=2;
		END_IF
	2:	(*FB_Power_On*)
		FB_CoupleAxis.Execute:=FALSE;
		FB_Power(On:=TRUE);
		fb_ton3.IN:=TRUE;
		State:=3;
	3:	(*wait*)
		FB_power();
		IF NOT FB_power.OnStatus THEN		(*FB_Power_OnÃ»ÓÐÖ´ÐÐÍê£¬wait£¬³¬Ê±FB Error*)
			IF NOT fb_ton3.Q THEN
				State:=3;
			ELSE
				ErrorID:=2;
				State:=99;
			END_IF
		ELSE
			State:=88;
		END_IF
	88:	(*All Done*)
		btn_PowerOn:=FALSE;
		State:=0;
		Error:=FALSE;
		ErrorID:=0;
		Busy:=FALSE;
		InitDone:=TRUE;

		FB_power.On:=FALSE;
		fb_ton1.IN:=FALSE;
		fb_ton2.IN:=FALSE;
		fb_ton3.IN:=FALSE;
		LED_Error:=FALSE;
	99:
		btn_PowerOn:=FALSE;
		State:=99;
		Error:=TRUE;
		Busy:=FALSE;
		InitDone:=FALSE;
		fb_ton1.IN:=FALSE;
		fb_ton2.IN:=FALSE;
		fb_ton3.IN:=FALSE;
		LED_Error:=TRUE;
END_CASE
END_ACTION

ACTION A_DecoupleAndPowerOff:
FB_DecoupleAxis();
CASE d_state OF
		0:(*Decouple*)
			FB_DecoupleAxis.Execute:=TRUE;
			FB_DecoupleAxis();
			d_state:=1;
		1:
			IF NOT FB_DecoupleAxis.OutGear THEN
				d_state:=1;
			ELSE
				d_state:=2;
			END_IF
		2:(*PowerOff*)
			FB_Power(Off:=TRUE);
				d_state:=3;
		3:
			IF NOT FB_power.OffStatus THEN
				d_state:=3;
			ELSE
				d_state:=88;
			END_IF
		88:(*ResetAllState*)
			btn_PowerOn:=FALSE;
			btn_GapMove:=FALSE;
			btn_GapStop:=FALSE;
			fb_ton1.IN:=FALSE;
			fb_ton2.IN:=FALSE;
			fb_ton3.IN:=FALSE;
			State:=0;
			Busy:=FALSE;
			InitDone:=FALSE;
			Error:=FALSE;
			ErrorID:=0;
			m_state:=0;
			s_state:=0;
			btn_PowerOff:=FALSE;
			d_state:=0;
			FB_DecoupleAxis.Execute:=FALSE;
			FB_DecoupleAxis.Reset:=TRUE;
			FB_DecoupleAxis();
			FB_CoupleAxis.Execute:=FALSE;
			FB_CoupleAxis.Reset:=TRUE;
			FB_CoupleAxis();
			Led_Run:=FALSE;
			Led_Error:=FALSE;
END_CASE
END_ACTION

ACTION A_MonitoringAllAxis:
(****************************************************************
NAME:			A_MonitoringAllAxis
DATA:			2017.2.24
VERSION:		1.0.0
DESCRIPTION:	
				Ã¿´ÎÑ­»·¾ùÖ´ÐÐÖáÎ»ÖÃºÍÖáÔË¶¯µÄ¼ì²é
				1.4ÖáÏà¶ÔÔË¶¯¼ì²é
				2.4Öá¹âÕ¤³ßÎ»ÖÃ¡¢ËÙ¶È¶Ô±È¼ì²é
				3.Ã¿Öá¹âÕ¤ºÍ±àÂëÆ÷Î»ÖÃ¶Ô±È¼ì²é
HISTORY:
				2017.2.24		NEW

***************************************************************)
(*************************************************************************************1.4ÖáÏà¶ÔÔË¶¯¼ì²é************************************************************************************)
(*1Öá¶¯£¬ÆäËüÈýÖá²»¶¯*)
IF  (LeftTopLin.Status.Moving AND NOT RightTopLin.Status.Moving AND NOT  LeftBottomLin.Status.Moving AND NOT RightBottomLin.Status.Moving)
	OR (NOT LeftTopLin.Status.Moving AND RightTopLin.Status.Moving AND NOT LeftBottomLin.Status.Moving AND NOT RightBottomLin.Status.Moving)
	OR (NOT LeftTopLin.Status.Moving AND NOT RightTopLin.Status.Moving AND LeftBottomLin.Status.Moving AND NOT  RightBottomLin.Status.Moving)
	OR (NOT LeftTopLin.Status.Moving AND NOT RightTopLin.Status.Moving AND NOT LeftBottomLin.Status.Moving AND RightBottomLin.Status.Moving) THEN
		btn_GapStop:=TRUE;
		FB_PlcEmergencyStop();
		Error:=TRUE;
		ErrorID:=11;
		LED_Error:=TRUE;
(*2Öá¶¯£¬2Öá²»¶¯*)
(*
ELSIF  (LeftTopLin.Status.Moving AND RightTopLin.Status.Moving AND NOT LeftBottomLin.Status.Moving AND NOT RightBottomLin.Status.Moving)
	OR  (LeftTopLin.Status.Moving AND NOT RightTopLin.Status.Moving AND LeftBottomLin.Status.Moving AND NOT RightBottomLin.Status.Moving)
	OR  (LeftTopLin.Status.Moving AND NOT RightTopLin.Status.Moving AND NOT LeftBottomLin.Status.Moving AND RightBottomLin.Status.Moving)
	OR  (NOT LeftTopLin.Status.Moving AND RightTopLin.Status.Moving AND LeftBottomLin.Status.Moving AND NOT RightBottomLin.Status.Moving)
	OR  (NOT LeftTopLin.Status.Moving AND RightTopLin.Status.Moving AND NOT LeftBottomLin.Status.Moving AND RightBottomLin.Status.Moving)
	OR  (NOT LeftTopLin.Status.Moving AND NOT RightTopLin.Status.Moving AND LeftBottomLin.Status.Moving AND RightBottomLin.Status.Moving) THEN
		btn_GapStop:=TRUE;
		FB_PlcEmergencyStop();
		Error:=TRUE;
		ErrorID:=12;
		LED_Error:=TRUE;
*)
(*3Öá¶¯£¬1Öá²»¶¯*)
ELSIF  (NOT LeftTopLin.Status.Moving AND RightTopLin.Status.Moving AND LeftBottomLin.Status.Moving AND RightBottomLin.Status.Moving)
	OR  (LeftTopLin.Status.Moving AND NOT RightTopLin.Status.Moving AND LeftBottomLin.Status.Moving AND RightBottomLin.Status.Moving)
	OR  (LeftTopLin.Status.Moving AND RightTopLin.Status.Moving AND NOT  LeftBottomLin.Status.Moving AND RightBottomLin.Status.Moving)
	OR  (LeftTopLin.Status.Moving AND RightTopLin.Status.Moving AND LeftBottomLin.Status.Moving AND NOT RightBottomLin.Status.Moving) THEN
		btn_GapStop:=TRUE;
		FB_PlcEmergencyStop();
		Error:=TRUE;
		ErrorID:=13;
		LED_Error:=TRUE;
END_IF
(*************************************************************************************2.4Öá¹âÕ¤³ßÎ»ÖÃ¡¢ËÙ¶È¶Ô±È¼ì²é**********************************************************************)
IF  st_Power<>0 THEN
(*Top Î»ÖÃºÍËÙ¶È±È¶Ô*)
		Diff_TopPos_actual:=Pos_leftTopLin-Pos_RightTopLin;
		Diff_TopVelo_actual:=Velo_leftTopLin-Velo_RightTopLin;
IF ABS(Pos_leftTopLin-Pos_RightTopLin)>Threshold_BCTopPos THEN
		btn_GapStop:=TRUE;
		FB_PlcEmergencyStop();
		Error:=TRUE;
		ErrorID:=14;
		LED_Error:=TRUE;
ELSIF ABS(Velo_leftTopLin-Velo_RightTopLin)>Threshold_BCTopVelo  THEN
		(*btn_GapStop:=TRUE;
		FB_PlcEmergencyStop();*)
		AA:=Velo_leftTopLin-Velo_RightTopLin;
		Error:=TRUE;
		ErrorID:=15;
(*Bottom Î»ÖÃºÍËÙ¶È±È¶Ô*)
ELSIF ABS(Pos_LeftBottomLin-Pos_RightBottomLin)>Threshold_BCBottomPos THEN
		btn_GapStop:=TRUE;
		FB_PlcEmergencyStop();
		Error:=TRUE;
		ErrorID:=16;
		LED_Error:=TRUE;
ELSIF ABS(Velo_leftBottomLin-Velo_RightBottomLin)>Threshold_BCBottomVelo  THEN
		(*btn_GapStop:=TRUE;
		FB_PlcEmergencyStop();*)
		BB:=Velo_leftBottomLin-Velo_RightBottomLin;
		Error:=TRUE;
		ErrorID:=17;
(*Left Î»ÖÃºÍËÙ¶È±È¶Ô*)
ELSIF ABS(Pos_LeftTopLin-Pos_LeftBottomLin)>Threshold_BCLeftPos  THEN
		btn_GapStop:=TRUE;
		FB_PlcEmergencyStop();
		Error:=TRUE;
		ErrorID:=18;
		LED_Error:=TRUE;
ELSIF  ABS(Velo_LeftTopLin-Velo_LeftBottomLin)>Threshold_BCLeftVelo THEN
		(*btn_GapStop:=TRUE;
		FB_PlcEmergencyStop();*)
		CC:=Velo_LeftTopLin-Velo_LeftBottomLin;
		Error:=TRUE;
		ErrorID:=19;
(*Right Î»ÖÃºÍËÙ¶È±È¶Ô*)
ELSIF ABS(Pos_RightTopLin-Pos_RightBottomLin)>Threshold_BCRightPos  THEN
		btn_GapStop:=TRUE;
		FB_PlcEmergencyStop();
		Error:=TRUE;
		ErrorID:=20;
		LED_Error:=TRUE;
ELSIF  ABS(Velo_RightTopLin-Velo_RightBottomLin)>Threshold_BCRightVelo THEN
		(*btn_GapStop:=TRUE;
		FB_PlcEmergencyStop();*)
		DD:=Velo_RightTopLin-Velo_RightBottomLin;
		Error:=TRUE;
		ErrorID:=21;
END_IF
END_IF
		LL:=Velo_LeftTopLin-Velo_LeftBottomLin;
		LL2:=Velo_RightTopLin-Velo_RightBottomLin;
(*********************************************************************************3.Ã¿Öá¹âÕ¤ºÍ±àÂëÆ÷Î»ÖÃ¶Ô±È¼ì²é**********************************************************************)
END_ACTION

ACTION A_PosDiffDetection:
IF ABS(PosDiff_LeftTopLin_actual-PosDiff_RightTopLin_actual)>0.2 THEN		(*ÉÏÖá×óÓÒÊµ¼ÊÎ»ÖÃÖ®²î*)
	ErrorID:=51;
	Error:=TRUE;
	btn_GapStop:=TRUE;
	FB_PlcEmergencyStop();
	LED_Error:=TRUE;
ELSIF ABS(PosDiff_LeftBottomLin_actual-PosDiff_RightBottomLin_actual)>0.2 THEN
	ErrorID:=53;
	Error:=TRUE;
	btn_GapStop:=TRUE;
	FB_PlcEmergencyStop();
	LED_Error:=TRUE;
END_IF
END_ACTION

END_PROGRAM

// ---- POUs/CommonFB/MainFB/FB_DecoupleAxis.TcPOU
(****************************************************************
NAME:			FB_DecoupleAxis
DATA:			2017.2.24
VERSION:		1.0.0
DESCRIPTION:	FB_DecoupleAxis
HISTORY:
				2017.2.16		NEW

***************************************************************)
FUNCTION_BLOCK FB_DecoupleAxis
VAR_INPUT
	Execute:BOOL;
	Reset:BOOL;
END_VAR
VAR_OUTPUT
	FbID:DINT:=1001;
	State:DINT;
	Busy:BOOL;
	OutGear:BOOL;
	Error:BOOL;
	ErrorID:DINT;
END_VAR
VAR
	Top_MC_GearOut: MC_GearOut;
	Bottom_MC_GearOut: MC_GearOut;
	fb_ton: TON;
END_VAR

IF Execute THEN
Busy:=TRUE;
fb_ton(PT:=t#0.1s);
CASE State OF
	0:	(*Decouple Check*)
		IF  LeftTopLin.NcToPlc.CoupleState=0 AND RightTopLin.NcToPlc.CoupleState=0
			AND LeftBottomLin.NcToPlc.CoupleState=0 AND RightBottomLin.NcToPlc.CoupleState=0 THEN	(*ÒÑ´¦ÓÚ·ÇñîºÏ£¬Ìø×ª88*)
			State:=88;
		ELSIF LeftTopLin.NcToPlc.CoupleState<>1 AND RightTopLin.NcToPlc.CoupleState<>3
			AND LeftBottomLin.NcToPlc.CoupleState<>1 AND RightBottomLin.NcToPlc.CoupleState<>3 THEN		(*´¦ÓÚ´íÎóµÄñîºÏ×´Ì¬£¬EStop*)
			ErrorID:=1;
			State:=-100;
		ELSIF Top_MC_GearOut.Error OR Bottom_MC_GearOut.Error THEN		(*FB ´íÎó*)
			ErrorID:=2;
			State:=99;
		ELSIF LeftTopLin.NcToPlc.CoupleState=1 AND RightTopLin.NcToPlc.CoupleState=3
			AND LeftBottomLin.NcToPlc.CoupleState=1 AND RightBottomLin.NcToPlc.CoupleState=3 THEN		(*Î¨Ò»ÕýÈ·µÄñîºÏ·½Ê½£¬×ªÏÂÒ»²½*)
			State:=1;
		END_IF
	1:	(*Decouple*)
		IF LeftTopLin.NcToPlc.CoupleState=1 AND RightTopLin.NcToPlc.CoupleState=3
			AND LeftBottomLin.NcToPlc.CoupleState=1 AND RightBottomLin.NcToPlc.CoupleState=3 THEN		(*ÔÙ´Î¼ì²éñîºÏ*)
			Top_MC_GearOut.Execute:=TRUE;
			Bottom_MC_GearOut.Execute:=TRUE;
			A_DecoupleMC();
			fb_ton.IN:=TRUE;
		ELSIF LeftTopLin.NcToPlc.CoupleState=0 AND RightTopLin.NcToPlc.CoupleState=0
			AND LeftBottomLin.NcToPlc.CoupleState=0 AND RightBottomLin.NcToPlc.CoupleState=0 THEN	(*ÒÑ´¦ÓÚ·ÇñîºÏ£¬Ìø×ª88*)
			State:=88;
		ELSE
			ErrorID:=3;
			State:=-100;
		END_IF
	2:	(*Decouple Wait*)
		A_DecoupleMC();
		IF NOT Top_MC_GearOut.Done OR NOT Bottom_MC_GearOut.Done THEN	(*ÓÐÒ»¸öGearOutÎ´Íê³É£¬¼ÌÐø¡£³¬Ê±Ôò±¨´í*)
			IF NOT fb_ton.Q THEN
				State:=2;
			ELSE
				ErrorID:=4;
				State:=99;
			END_IF
		ELSIF Top_MC_GearOut.Done AND Bottom_MC_GearOut.Done
			AND LeftTopLin.NcToPlc.CoupleState=0 AND RightTopLin.NcToPlc.CoupleState=0
			AND LeftBottomLin.NcToPlc.CoupleState=0 AND RightBottomLin.NcToPlc.CoupleState=0 THEN		(*Decouple DoneÇÒñîºÏ×´Ì¬ÕýÈ·£¬×ª88*)
			State:=88;
		ELSE
			ErrorID:=5;
			State:=-100;
		END_IF
	88:	(*Done*)
		Execute:=FALSE;
		State:=0;
		Busy:=FALSE;
		OutGear:=TRUE;
		Error:=FALSE;
		ErrorID:=0;
		Top_MC_GearOut.Execute:=FALSE;
		Bottom_MC_GearOut.Execute:=FALSE;
		A_DecoupleMC();
		fb_ton.IN:=FALSE;
	99:	(*FB Error*)
		Execute:=FALSE;
		State:=99;
		Busy:=FALSE;
		OutGear:=FALSE;
		Error:=TRUE;
		Top_MC_GearOut.Execute:=FALSE;
		Bottom_MC_GearOut.Execute:=FALSE;
		A_DecoupleMC();
		fb_ton.IN:=FALSE;
	-100:	(*EStop Error*)
		FB_PlcEmergencyStop();
		Execute:=FALSE;
		State:=-100;
		Busy:=FALSE;
		OutGear:=FALSE;
		Error:=TRUE;
		Top_MC_GearOut.Execute:=FALSE;
		Bottom_MC_GearOut.Execute:=FALSE;
		A_DecoupleMC();
		fb_ton.IN:=FALSE;

END_CASE
END_IF
IF Reset THEN
		Execute:=FALSE;
		State:=0;
		Busy:=FALSE;
		OutGear:=FALSE;
		Error:=FALSE;
		ErrorID:=0;
		Top_MC_GearOut.Execute:=FALSE;
		Bottom_MC_GearOut.Execute:=FALSE;
		A_DecoupleMC();
		fb_ton.IN:=FALSE;
		Reset:=FALSE;
END_IF

ACTION A_DecoupleMC:
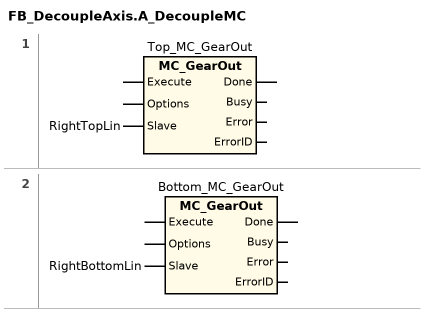
// NETWORK 1
Top_MC_GearOut(Slave := RightTopLin); // MC_GearOut

// NETWORK 2
Bottom_MC_GearOut(Slave := RightBottomLin); // MC_GearOut
END_ACTION

END_FUNCTION_BLOCK

// ---- POUs/2.SingleMotorMode/DebugMode/DebugMode.TcPOU
PROGRAM DebugMode
VAR
(* Common*)
	d_state: DINT;(*PowerOffState*)
	InitDone:BOOL;
	Busy: BOOL;
	fb_ton: TON;
	PowerState: INT;(*PowerOnState*)
	ton_t: TON;
(*Key Command*)
	btn_PowerOn: BOOL;
	btn_PowerOff: BOOL;
	LeftTopLinPositionNew:LREAL;
	LeftTopLinVelocityNew:LREAL:=1;
	btn_LeftTopLinMove:BOOL;
	btn_LeftTopLinStop:BOOL;
	RightTopLinPositionNew:LREAL;
	RightTopLinVelocityNew:LREAL:=1;
	btn_RightTopLinMove:BOOL;
	btn_RightTopLinStop:BOOL;
	LeftBottomLinPositionNew:LREAL;
	LeftBottomLinVelocityNew:LREAL:=1;
	btn_LeftBottomLinMove:BOOL;
	btn_LeftBottomLinStop:BOOL;
	RightBottomLinPositionNew:LREAL;
	RightBottomLinVelocityNew:LREAL:=1;
	btn_RightBottomLinMove:BOOL;
	btn_RightBottomLinStop:BOOL;
(*LeftTopLin*)
	fb_ton1_1:TON;
	fb_ton1_2:TON;
	LeftTopLinState:DINT;
	LeftTopLinBusy:BOOL;
	LeftTopLin_m_state: DINT;
	LeftTopLin_s_state: DINT;
(*RightTopLin*)
	fb_ton2_1:TON;
	fb_ton2_2:TON;
	RightTopLinState:DINT;
	RightTopLinBusy:BOOL;
	RightTopLin_m_state: DINT;
	RightTopLin_s_state: DINT;
(*LeftBottomLin*)
	fb_ton3_1:TON;
	fb_ton3_2:TON;
	LeftBottomLinState:DINT;
	LeftBottomLinBusy:BOOL;
	LeftBottomLin_m_state: DINT;
	LeftBottomLin_s_state: DINT;
(*RightBottomLin*)
	fb_ton4_1:TON;
	fb_ton4_2:TON;
	RightBottomLinState:DINT;
	RightBottomLinBusy:BOOL;
	RightBottomLin_m_state: DINT;
	RightBottomLin_s_state: DINT;


	btn_LeftTopStop: BOOL;
	(*¼ì²âµ½ÏÞÎ»£¬»Ö¸´Move×´Ì¬*)
	FTrig_ReachLS: F_TRIG;
	FTrig_btn_GapMove: F_TRIG;
	btn_Power: BOOL;
END_VAR

(*********************************************************************Monitor All Carrirt Position***********************************************)
A_MonitoringAllAxis();
(*********************************************************************A_PosDiffDetection***********************************************)
A_PosDiffDetection();
(*********************************************************************btn_PowerOn************************************************************)
IF btn_Power AND st_Power=0 THEN
	btn_PowerOn:=TRUE;
	btn_Power:=FALSE;
END_IF
IF btn_Power AND st_Power=1 THEN
	btn_PowerOff:=TRUE;
	btn_Power:=FALSE;
END_IF
(*********************************************************************btn_PowerOn************************************************************)
IF btn_PowerOn THEN
	A_PowerOn();
END_IF
(******************************************************ÉÏµç×´Ì¬£¬´¦ÓÚñîºÏ×´Ì¬£¬ESTOP***********************************************)
IF NOT btn_PowerOff THEN
	IF st_Power=1 AND st_Couple<>0THEN
		Error:=TRUE;
		ErrorID:=101;
		FB_PlcEmergencyStop();
		LED_Error:=TRUE;
	END_IF
END_IF
(*********************************************************************LeftTop_MOVE*****************************************************************)
IF InitDone THEN
	IF btn_LeftTopLinMove THEN
		CASE LeftTopLin_m_state OF
			0:
				FB_Move.Mode:=4;						(*1£ºgapÄ£Ê½£»2£ºµ¥ÁºÄ£Ê½£¬3£ºtaperÄ£Ê½£¬4£ºDebugÄ£Ê½*)
				FB_Move.CoupleState:=st_Couple;			(*ñîºÏ×´Ì¬ÊäÈë*)
				FB_Move.PowerState:=st_Power;			(*µçÔ´×´Ì¬ÊäÈë*)
				FB_Move.LeftTopMove:=TRUE;				(*Execute TRUE*)
				FB_Move.LeftTopPosition:=LeftTopLinPositionNew;	(*Î»ÖÃ*)
				FB_Move.LeftTopVelocity:=LeftTopLinVelocityNew;	(*ËÙ¶È*)
				FB_Move();								(*Æô¶¯FB*)
				LeftTopLin_m_state:=1;
			1:
				FB_Move();
				IF NOT FB_Move.LeftTopDone THEN			(*ÔË¶¯Î´Íê³É£¬Ñ­»·*)
					LeftTopLin_m_state:=1;
					LED_Run:=TRUE;
				ELSE									(*ÔË¶¯Íê³É£¬ÏÂÒ»²½*)
					LeftTopLin_m_state:=88;
				END_IF

			88:
				btn_LeftTopLinMove:=FALSE;					(*×´Ì¬»Ö¸´*)
				LeftTopLin_m_state:=0;
				LED_Run:=FALSE;
		END_CASE
	END_IF
END_IF
(*******************************************************************LeftTop_STOP********************************************************************)
IF btn_LeftTopLinStop THEN
	LED_Run:=FALSE;
	FB_Move.LeftTopReset:=TRUE;							(*¸øÔË¶¯FB¸øÍ£Ö¹ÐÅºÅ£¬Ê¹FB_Move×´Ì¬»Ö¸´*)
	FB_Move();											(*Æô¶¯FB_Move*)
	btn_LeftTopLinMove:=FALSE;							(*btn_GapMove:=FALSE*)
	LeftTopLin_m_state:=0;											(*m_state:=0;*)
	CASE LeftTopLin_s_state OF
			0:
				FB_Stop.Mode:=4;							(*1£ºgapÄ£Ê½£»2£ºµ¥ÁºÄ£Ê½£»3£ºtaperÄ£Ê½*)
				FB_Stop.CoupleState:=st_Couple;			(*ñîºÏ×´Ì¬ÊäÈë*)
				FB_Stop.PowerState:=st_Power;				(*µçÔ´×´Ì¬ÊäÈë*)
				FB_Stop.LeftTopStop:=TRUE;				(*Execute TRUE*)
				FB_Stop();								(*Æô¶¯FB*)
				LeftTopLin_s_state:=1;
			1:
				FB_Stop();
				IF NOT FB_Stop.LeftTopDone THEN			(*Í£Ö¹Î´Íê³É£¬Ñ­»·*)
					LeftTopLin_s_state:=1;
				ELSE									(*Í£Ö¹Íê³É£¬ÏÂÒ»²½*)
					LeftTopLin_s_state:=88;
				END_IF
			88:
				btn_LeftTopLinStop:=FALSE;						(*»Ö¸´×´Ì¬*)
				FB_Move.LeftTopReset:=FALSE;					(*ÔËÐÐFB*)
				LeftTopLin_s_state:=0;
		END_CASE

END_IF
(*********************************************************************RightTop_MOVE*****************************************************************)
IF InitDone THEN
	IF btn_RightTopLinMove THEN
		CASE RightTopLin_m_state OF
			0:
				FB_Move.Mode:=4;						(*1£ºgapÄ£Ê½£»2£ºµ¥ÁºÄ£Ê½£¬3£ºtaperÄ£Ê½£¬4£ºDebugÄ£Ê½*)
				FB_Move.CoupleState:=st_Couple;			(*ñîºÏ×´Ì¬ÊäÈë*)
				FB_Move.PowerState:=st_Power;			(*µçÔ´×´Ì¬ÊäÈë*)
				FB_Move.RightTopMove:=TRUE;				(*Execute TRUE*)
				FB_Move.RightTopPosition:=RightTopLinPositionNew;	(*Î»ÖÃ*)
				FB_Move.RightTopVelocity:=RightTopLinVelocityNew;	(*ËÙ¶È*)
				FB_Move();								(*Æô¶¯FB*)
				RightTopLin_m_state:=1;
			1:
				FB_Move();
				IF NOT FB_Move.RightTopDone THEN			(*ÔË¶¯Î´Íê³É£¬Ñ­»·*)
					RightTopLin_m_state:=1;
					LED_Run:=TRUE;
				ELSE									(*ÔË¶¯Íê³É£¬ÏÂÒ»²½*)
					RightTopLin_m_state:=88;
				END_IF

			88:
				btn_RightTopLinMove:=FALSE;					(*×´Ì¬»Ö¸´*)
				RightTopLin_m_state:=0;
				LED_Run:=FALSE;
		END_CASE
	END_IF
END_IF
(*******************************************************************RightTop_STOP********************************************************************)
IF btn_RightTopLinStop THEN
	LED_Run:=FALSE;
	FB_Move.RightTopReset:=TRUE;							(*¸øÔË¶¯FB¸øÍ£Ö¹ÐÅºÅ£¬Ê¹FB_Move×´Ì¬»Ö¸´*)
	FB_Move();											(*Æô¶¯FB_Move*)
	btn_RightTopLinMove:=FALSE;							(*btn_GapMove:=FALSE*)
	RightTopLin_m_state:=0;											(*m_state:=0;*)
	CASE RightTopLin_s_state OF
			0:
				FB_Stop.Mode:=4;							(*1£ºgapÄ£Ê½£»2£ºµ¥ÁºÄ£Ê½£»3£ºtaperÄ£Ê½*)
				FB_Stop.CoupleState:=st_Couple;			(*ñîºÏ×´Ì¬ÊäÈë*)
				FB_Stop.PowerState:=st_Power;				(*µçÔ´×´Ì¬ÊäÈë*)
				FB_Stop.RightTopStop:=TRUE;				(*Execute TRUE*)
				FB_Stop();								(*Æô¶¯FB*)
				RightTopLin_s_state:=1;
			1:
				FB_Stop();
				IF NOT FB_Stop.RightTopDone THEN			(*Í£Ö¹Î´Íê³É£¬Ñ­»·*)
					RightTopLin_s_state:=1;
				ELSE									(*Í£Ö¹Íê³É£¬ÏÂÒ»²½*)
					RightTopLin_s_state:=88;
				END_IF
			88:
				btn_RightTopLinStop:=FALSE;						(*»Ö¸´×´Ì¬*)
				FB_Move.RightTopReset:=FALSE;					(*ÔËÐÐFB*)
				RightTopLin_s_state:=0;
		END_CASE

END_IF
(*********************************************************************LeftBottom_MOVE*****************************************************************)
IF InitDone THEN
	IF btn_LeftBottomLinMove THEN
		CASE LeftBottomLin_m_state OF
			0:
				FB_Move.Mode:=4;						(*1£ºgapÄ£Ê½£»2£ºµ¥ÁºÄ£Ê½£¬3£ºtaperÄ£Ê½£¬4£ºDebugÄ£Ê½*)
				FB_Move.CoupleState:=st_Couple;			(*ñîºÏ×´Ì¬ÊäÈë*)
				FB_Move.PowerState:=st_Power;			(*µçÔ´×´Ì¬ÊäÈë*)
				FB_Move.LeftBottomMove:=TRUE;				(*Execute TRUE*)
				FB_Move.LeftBottomPosition:=LeftBottomLinPositionNew;	(*Î»ÖÃ*)
				FB_Move.LeftBottomVelocity:=LeftBottomLinVelocityNew;	(*ËÙ¶È*)
				FB_Move();								(*Æô¶¯FB*)
				LeftBottomLin_m_state:=1;
			1:
				FB_Move();
				IF NOT FB_Move.LeftBottomDone THEN			(*ÔË¶¯Î´Íê³É£¬Ñ­»·*)
					LeftBottomLin_m_state:=1;
					LED_Run:=TRUE;
				ELSE									(*ÔË¶¯Íê³É£¬ÏÂÒ»²½*)
					LeftBottomLin_m_state:=88;
				END_IF

			88:
				btn_LeftBottomLinMove:=FALSE;					(*×´Ì¬»Ö¸´*)
				LeftBottomLin_m_state:=0;
				LED_Run:=FALSE;
		END_CASE
	END_IF
END_IF
(*******************************************************************LeftBottom_STOP********************************************************************)
IF btn_LeftBottomLinStop THEN
	LED_Run:=FALSE;
	FB_Move.LeftBottomReset:=TRUE;							(*¸øÔË¶¯FB¸øÍ£Ö¹ÐÅºÅ£¬Ê¹FB_Move×´Ì¬»Ö¸´*)
	FB_Move();											(*Æô¶¯FB_Move*)
	btn_LeftBottomLinMove:=FALSE;							(*btn_GapMove:=FALSE*)
	LeftBottomLin_m_state:=0;											(*m_state:=0;*)
	CASE LeftBottomLin_s_state OF
			0:
				FB_Stop.Mode:=4;							(*1£ºgapÄ£Ê½£»2£ºµ¥ÁºÄ£Ê½£»3£ºtaperÄ£Ê½*)
				FB_Stop.CoupleState:=st_Couple;			(*ñîºÏ×´Ì¬ÊäÈë*)
				FB_Stop.PowerState:=st_Power;				(*µçÔ´×´Ì¬ÊäÈë*)
				FB_Stop.LeftBottomStop:=TRUE;				(*Execute TRUE*)
				FB_Stop();								(*Æô¶¯FB*)
				LeftBottomLin_s_state:=1;
			1:
				FB_Stop();
				IF NOT FB_Stop.LeftBottomDone THEN			(*Í£Ö¹Î´Íê³É£¬Ñ­»·*)
					LeftBottomLin_s_state:=1;
				ELSE									(*Í£Ö¹Íê³É£¬ÏÂÒ»²½*)
					LeftBottomLin_s_state:=88;
				END_IF
			88:
				btn_LeftBottomLinStop:=FALSE;						(*»Ö¸´×´Ì¬*)
				FB_Move.LeftBottomReset:=FALSE;					(*ÔËÐÐFB*)
				LeftBottomLin_s_state:=0;
		END_CASE

END_IF

(*********************************************************************RightTop_MOVE*****************************************************************)
IF InitDone THEN
	IF btn_RightBottomLinMove THEN
		CASE RightBottomLin_m_state OF
			0:
				FB_Move.Mode:=4;						(*1£ºgapÄ£Ê½£»2£ºµ¥ÁºÄ£Ê½£¬3£ºtaperÄ£Ê½£¬4£ºDebugÄ£Ê½*)
				FB_Move.CoupleState:=st_Couple;			(*ñîºÏ×´Ì¬ÊäÈë*)
				FB_Move.PowerState:=st_Power;			(*µçÔ´×´Ì¬ÊäÈë*)
				FB_Move.RightBottomMove:=TRUE;				(*Execute TRUE*)
				FB_Move.RightBottomPosition:=RightBottomLinPositionNew;	(*Î»ÖÃ*)
				FB_Move.RightBottomVelocity:=RightBottomLinVelocityNew;	(*ËÙ¶È*)
				FB_Move();								(*Æô¶¯FB*)
				RightBottomLin_m_state:=1;
			1:
				FB_Move();
				IF NOT FB_Move.RightBottomDone THEN			(*ÔË¶¯Î´Íê³É£¬Ñ­»·*)
					RightBottomLin_m_state:=1;
					LED_Run:=TRUE;
				ELSE									(*ÔË¶¯Íê³É£¬ÏÂÒ»²½*)
					RightBottomLin_m_state:=88;
				END_IF

			88:
				btn_RightBottomLinMove:=FALSE;					(*×´Ì¬»Ö¸´*)
				RightBottomLin_m_state:=0;
				LED_Run:=FALSE;
		END_CASE
	END_IF
END_IF
(*******************************************************************RightBottom_STOP********************************************************************)
IF btn_RightBottomLinStop THEN
	LED_Run:=FALSE;
	FB_Move.RightBottomReset:=TRUE;							(*¸øÔË¶¯FB¸øÍ£Ö¹ÐÅºÅ£¬Ê¹FB_Move×´Ì¬»Ö¸´*)
	FB_Move();											(*Æô¶¯FB_Move*)
	btn_RightBottomLinMove:=FALSE;							(*btn_GapMove:=FALSE*)
	RightBottomLin_m_state:=0;											(*m_state:=0;*)
	CASE RightBottomLin_s_state OF
			0:
				FB_Stop.Mode:=4;							(*1£ºgapÄ£Ê½£»2£ºµ¥ÁºÄ£Ê½£»3£ºtaperÄ£Ê½*)
				FB_Stop.CoupleState:=st_Couple;			(*ñîºÏ×´Ì¬ÊäÈë*)
				FB_Stop.PowerState:=st_Power;				(*µçÔ´×´Ì¬ÊäÈë*)
				FB_Stop.RightBottomStop:=TRUE;				(*Execute TRUE*)
				FB_Stop();								(*Æô¶¯FB*)
				RightBottomLin_s_state:=1;
			1:
				FB_Stop();
				IF NOT FB_Stop.RightBottomDone THEN			(*Í£Ö¹Î´Íê³É£¬Ñ­»·*)
					RightBottomLin_s_state:=1;
				ELSE									(*Í£Ö¹Íê³É£¬ÏÂÒ»²½*)
					RightBottomLin_s_state:=88;
				END_IF
			88:
				btn_RightBottomLinStop:=FALSE;						(*»Ö¸´×´Ì¬*)
				FB_Move.RightBottomReset:=FALSE;					(*ÔËÐÐFB*)
				RightBottomLin_s_state:=0;
		END_CASE

END_IF
(*********************************************************************btn_PowerOff************************************************************)
IF btn_PowerOff THEN
	A_PowerOff();
END_IF
(****************************MoveIndicator***************************)
IF Velo_LeftTopLin>0 THEN
	LeftTopLinMoveIndicator:=1;
ELSIF Velo_LeftTopLin<0 THEN
	LeftTopLinMoveIndicator:=-1;
ELSE
	LeftTopLinMoveIndicator:=0;
END_IF
IF Velo_RightTopLin>0 THEN
	RightTopLinMoveIndicator:=1;
ELSIF Velo_RightTopLin<0 THEN
	RightTopLinMoveIndicator:=-1;
ELSE
	RightTopLinMoveIndicator:=0;
END_IF
IF Velo_LeftBottomLin>0 THEN
	LeftBottomLinMoveIndicator:=1;
ELSIF Velo_LeftBottomLin<0 THEN
	LeftBottomLinMoveIndicator:=-1;
ELSE
	LeftBottomLinMoveIndicator:=0;
END_IF
IF Velo_RightBottomLin>0 THEN
	RightBottomLinMoveIndicator:=1;
ELSIF Velo_RightBottomLin<0 THEN
	RightBottomLinMoveIndicator:=-1;
ELSE
	RightBottomLinMoveIndicator:=0;
END_IF
(*********************************************************************ÏÞÎ»Åö´¥×´Ì¬»Ö¸´************************************************************)
(*Èç¹û¼ì²âµ½ÏØÏÞÎ»¿ª¹ØÏÂ½µÑØ£¬»Ö¸´Move×´Ì¬*)
FTrig_ReachLS(CLK:=Unreach_LS_Top AND Unreach_LS_Bottom);
IF FTrig_ReachLS.Q THEN
	btn_LeftTopLinStop:=TRUE;
	btn_RightTopLinStop:=TRUE;
	btn_LeftBottomLinStop:=TRUE;
	btn_RightBottomLinStop:=TRUE;
END_IF
IF btn_LeftTopLinStop THEN
	btn_RightTopLinStop:=TRUE;
END_IF
IF btn_RightTopLinStop THEN
	btn_LeftBottomLinStop:=TRUE;
END_IF
IF btn_LeftBottomLinStop THEN
	btn_RightBottomLinStop:=TRUE;
END_IF

(*Èç¹û¼ì²âµ½TopÏÞÎ»¿ª¹ØFALSE£¬ÇÒÄ¿±êÎ»ÖÃ´óÓÚµ±Ç°Î»ÖÃÊ±£¬»òÕßÏà·´Ê±£¬»Ö¸´Move×´Ì¬*)
IF NOT Unreach_LS_Top AND LeftTopLinPositionNew-Pos_LeftTopLin>0.0005 AND btn_LeftTopLinMove THEN
	btn_LeftTopLinStop:=TRUE;
END_IF
IF NOT Unreach_LS_Bottom AND RightTopLinPositionNew-Pos_RightTopLin<0.0005 AND btn_RightTopLinMove THEN
	btn_RightTopLinStop:=TRUE;
END_IF
IF NOT Unreach_LS_Top AND LeftBottomLinPositionNew-Pos_LeftBottomLin>0.0005 AND btn_LeftBottomLinMove THEN
	btn_LeftBottomLinStop:=TRUE;
END_IF
IF NOT Unreach_LS_Bottom AND RightBottomLinPositionNew-Pos_RightBottomLin<0.0005 AND btn_RightBottomLinMove THEN
	btn_RightBottomLinStop:=TRUE;
END_IF

ACTION A_monitoringAllAxis:
(****************************************************************
NAME:			A_MonitoringAllAxis
DATA:			2017.5.8
VERSION:		1.0.0
DESCRIPTION:	
				Ã¿´ÎÑ­»·¾ùÖ´ÐÐÖáÎ»ÖÃºÍÖáÔË¶¯µÄ¼ì²é
				1.4ÖáÏà¶ÔÔË¶¯¼ì²é
				2.4Öá¹âÕ¤³ßÎ»ÖÃ¡¢ËÙ¶È¶Ô±È¼ì²é
				3.Ã¿Öá¹âÕ¤ºÍ±àÂëÆ÷Î»ÖÃ¶Ô±È¼ì²é
HISTORY:
				2017.5.8	NEW

***************************************************************)
(*************************************************************************************1.4ÖáÏà¶ÔÔË¶¯¼ì²é************************************************************************************)
(*DebugÄ£Ê½£¬Öá¾ù×ÔÓÉ»î¶¯*)
(*(*³ýÁËÓÒÉÏºÍÓÒÏÂÖáÒ»Æð¶¯£¬ÆäÓàÖá¶¯¶¼ESTOP*)
(*×óÉÏ¡¢×óÏÂÖá¶¯*)
IF  LeftTopLin.Status.Moving OR LeftBottomLin.Status.Moving THEN
	FB_PlcEmergencyStop();
	Error:=TRUE;
	ErrorID:=11;
END_IF
(*ÓÒÉÏ¶¯¡¢ÓÒÏÂ²»¶¯£¬»òÕßÓÒÏÂ¶¯¡¢ÓÒÉÏ²»¶¯¡£ESTOP*)
IF (RightTopLin.Status.Moving AND RightBottomLin.Status.NotMoving) OR (RightTopLin.Status.NotMoving AND RightBottomLin.Status.Moving) THEN
		FB_PlcEmergencyStop();
		Error:=TRUE;
		ErrorID:=12;
END_IF
*)
(*************************************************************************************2.4Öá¹âÕ¤³ßÎ»ÖÃ¡¢ËÙ¶È¶Ô±È¼ì²é**********************************************************************)
IF st_power<>0 THEN
(*×óÖáÉÏÏÂÎ»ÖÃ¶Ô±È£¬³¬³öESTOP*)
IF ABS(Pos_LeftTopLin-Pos_LeftBottomLin)>Threshold_LeftPos_Debug  THEN
		btn_LeftTopLinStop:=TRUE;
		btn_RightTopLinStop:=TRUE;
		btn_LeftBottomLinStop:=TRUE;
		btn_RightBottomLInStop:=TRUE;
		FB_PlcEmergencyStop();
		Error:=TRUE;
		ErrorID:=11;
		LED_Error:=TRUE;
END_IF
(*ÓÒÖáÉÏÏÂÎ»ÖÃËÙ¶È¶Ô±È£¬³¬³öESTOP*)
IF ABS(Pos_RightTopLin-Pos_RightBottomLin)>Threshold_RightPos_Debug  THEN
		btn_LeftTopLinStop:=TRUE;
		btn_RightTopLinStop:=TRUE;
		btn_LeftBottomLinStop:=TRUE;
		btn_RightBottomLInStop:=TRUE;
		FB_PlcEmergencyStop();
		Error:=TRUE;
		ErrorID:=12;
		LED_Error:=TRUE;
END_IF
(*ÉÏÖá×óÓÒÎ»ÖÃ¶Ô±È£¬³¬³öESTOP*)
IF ABS(Pos_LeftTopLin-Pos_RightTopLin)>Threshold_TopPos_Debug  THEN
		btn_LeftTopLinStop:=TRUE;
		btn_RightTopLinStop:=TRUE;
		btn_LeftBottomLinStop:=TRUE;
		btn_RightBottomLInStop:=TRUE;
		FB_PlcEmergencyStop();
		Error:=TRUE;
		ErrorID:=13;
		LED_Error:=TRUE;
END_IF
(*ÏÂÖá×óÓÒÎ»ÖÃ¶Ô±È£¬³¬³öESTOP*)
IF ABS(Pos_LeftBottomLin-Pos_RightBottomLin)>Threshold_BottomPos_Debug  THEN
		btn_LeftTopLinStop:=TRUE;
		btn_RightTopLinStop:=TRUE;
		btn_LeftBottomLinStop:=TRUE;
		btn_RightBottomLInStop:=TRUE;
		FB_PlcEmergencyStop();
		Error:=TRUE;
		ErrorID:=14;
		LED_Error:=TRUE;
END_IF
END_IF
(*********************************************************************************3.Ã¿Öá¹âÕ¤ºÍ±àÂëÆ÷Î»ÖÃ¶Ô±È¼ì²é**********************************************************************)
END_ACTION

ACTION A_PosDiffDetection:
IF ABS(PosDiff_LeftTopLin_actual-PosDiff_RightTopLin_actual)>0.2 THEN
	ErrorID:=51;
	Error:=TRUE;
	btn_LeftTopLinStop:=TRUE;
	btn_RightTopLinStop:=TRUE;
	btn_LeftBottomLinStop:=TRUE;
	btn_RightBottomLInStop:=TRUE;
	FB_PlcEmergencyStop();
	LED_Error:=TRUE;
ELSIF ABS(PosDiff_LeftBottomLin_actual-PosDiff_RightBottomLin_actual)>0.2 THEN
	ErrorID:=53;
	Error:=TRUE;
	btn_LeftTopLinStop:=TRUE;
	btn_RightTopLinStop:=TRUE;
	btn_LeftBottomLinStop:=TRUE;
	btn_RightBottomLInStop:=TRUE;
	FB_PlcEmergencyStop();
	LED_Error:=TRUE;
END_IF
END_ACTION

ACTION A_PowerOff:
CASE d_state OF
		0:(*PowerOff*)
			FB_Power(Off:=TRUE);
				d_state:=1;
		1:
			IF NOT FB_power.OffStatus THEN
				d_state:=1;
			ELSE
				d_state:=88;
			END_IF
		88:(*ResetAllState*)
			btn_PowerOn:=FALSE;
			btn_PowerOff:=FALSE;
			ton_t.IN:=FALSE;
			InitDone:=FALSE;
			Error:=FALSE;
			ErrorID:=0;
			d_state:=0;

			btn_LeftTopLinMove:=FALSE;
			btn_LeftTopLinStop:=FALSE;
			fb_ton1_1.IN:=FALSE;
			fb_ton1_2.IN:=FALSE;
			LeftTopLinState:=0;
			LeftTopLinBusy:=FALSE;
			LeftTopLin_m_state:=0;
			LeftTopLin_s_state:=0;

			btn_RightTopLinMove:=FALSE;
			btn_RightTopLinStop:=FALSE;
			fb_ton2_1.IN:=FALSE;
			fb_ton2_2.IN:=FALSE;
			RightTopLinState:=0;
			RightTopLinBusy:=FALSE;
			RightTopLin_m_state:=0;
			RightTopLin_s_state:=0;

			btn_LeftBottomLinMove:=FALSE;
			btn_LeftBottomLinStop:=FALSE;
			fb_ton3_1.IN:=FALSE;
			fb_ton3_2.IN:=FALSE;
			LeftBottomLinState:=0;
			LeftBottomLinBusy:=FALSE;
			LeftBottomLin_m_state:=0;
			LeftBottomLin_s_state:=0;

			btn_RightBottomLinMove:=FALSE;
			btn_RightBottomLinStop:=FALSE;
			fb_ton4_1.IN:=FALSE;
			fb_ton4_2.IN:=FALSE;
			RightBottomLinState:=0;
			RightBottomLinBusy:=FALSE;
			RightBottomLin_m_state:=0;
			RightBottomLin_s_state:=0;

		LED_Error:=FALSE;
		LED_Run:=FALSE;

END_CASE
END_ACTION

ACTION A_PowerOn:
(****************************************************************
NAME:			A_SetAxisPositionAndPowerOn
DATA:			2017.3.27
VERSION:		1.0.0
DESCRIPTION:	
				ÉÏµãÃüÁîºó£¬Ë³ÐòÖ´ÐÐ£º
				1.FB_SetAxisPosition
				2.FB_PowerOn
				·µ»ØÖ´ÐÐÊÇ·ñ³É¹¦
HISTORY:
				2017.3.27		NEW
				2017.5.8		É¾³ýÁËsetAxisPosition£¬ÒÆ¶¯µ½MAIN³ÌÐòÖÐ
							±ä¸üNAMEÎªA_PowerOn

***************************************************************)
fb_ton(PT:=t#0.5s);
CASE PowerState OF
	0:	(*FB_Power_On*)
		FB_Power(On:=TRUE);
		fb_ton.IN:=TRUE;
		PowerState:=1;
	1:	(*wait*)
		FB_power();
		IF NOT FB_power.OnStatus THEN		(*FB_Power_OnÃ»ÓÐÖ´ÐÐÍê£¬wait£¬³¬Ê±FB Error*)
			IF NOT fb_ton.Q THEN
				PowerState:=1;
			ELSE
				ErrorID:=1;
				PowerState:=99;
			END_IF
		ELSE
			PowerState:=88;
		END_IF
	88:	(*All Done*)
		btn_PowerOn:=FALSE;
		PowerState:=0;
		Error:=FALSE;
		ErrorID:=0;
		Busy:=FALSE;
		InitDone:=TRUE;
		FB_power.On:=FALSE;
		fb_ton.IN:=FALSE;
	99:
		btn_PowerOn:=FALSE;
		PowerState:=99;
		Error:=TRUE;
		Busy:=FALSE;
		InitDone:=FALSE;
		FB_Power.On:=FALSE;
		fb_ton.IN:=FALSE;
		LED_Error:=TRUE;
END_CASE
END_ACTION

END_PROGRAM

// ---- POUs/1.CarrierMode/GapMode/BCGapMode.TcPOU
PROGRAM BCGapMode
VAR
	(*key Command*)
	btn_Power:BOOL;
	btn_PowerOn: BOOL;
	btn_PowerOff: BOOL;
(*GapMode*)
	BCGapPositionNew:LREAL:=20;
	BCGapVelocityNew:LREAL:=1;
	BCGapPositionDisplay:LREAL;
	BCGapVelocityDisplay:LREAL;
	btn_BCGapMove:BOOL;
	btn_BCGapStop:BOOL;
	(*Var*)
	fb_ton1:TON;
	fb_ton2:TON;
	fb_ton3:TON;
	(*Status*)
	State:DINT;
	Busy:BOOL;
	InitPowerDone:BOOL;
	InitCompensationDatasDone:BOOL;
	(*FB*)
	m_state: DINT;
	s_state: DINT;
	(*¼ì²âµ½ÏÞÎ»£¬»Ö¸´Move×´Ì¬*)
	FTrig_ReachLS: F_TRIG;
	FTrig_btn_GapMove: F_TRIG;
	GapOutRange: BOOL;
	(*PowerOff*)
	d_state: DINT;
	i: INT;
	j: INT;
	moni_State:DINT;
END_VAR

BCGapPositionDisplay:=(LeftTopLinPositionDisplay+RightTopLinPositionDisplay+LeftBottomLinPositionDisplay+RightBottomLinPositionDisplay)/2;
BCGapVelocityDisplay:=(LeftTopLinVelocityDisplay+RightTopLinVelocityDisplay+LeftBottomLinVelocityDisplay+RightBottomLinVelocityDisplay)/2;
(*********************************************************************btn_PowerOn************************************************************)
IF btn_Power AND st_Power=0 THEN
	btn_PowerOn:=TRUE;
	btn_Power:=FALSE;
END_IF
IF btn_Power AND st_Power=1 THEN
	btn_PowerOff:=TRUE;
	btn_Power:=FALSE;
END_IF
//
IF btn_PowerOn THEN
	A_PowerOn();
END_IF
(******************************************************ÉÏµç×´Ì¬£¬´¦ÓÚñîºÏ×´Ì¬£¬ESTOP***********************************************)
IF NOT btn_PowerOff THEN
	IF st_Power=1 AND st_Couple<>0THEN
		Error:=TRUE;
		ErrorID:=101;
		LeftTopLinMoveIndicator:=0;
		RightTopLinMoveIndicator:=0;
		LeftBottomLinMoveIndicator:=0;
		RightBottomLinMoveIndicator:=0;
		FB_PlcEmergencyStop();
		LED_Error:=TRUE;
	END_IF
END_IF
(*********************************************************************Monitor All Carrirt Position***********************************************)
A_MonitoringAllAxis();
(*********************************************************************A_PosDiffDetection***********************************************)
A_PosDiffDetection();
(*****************************************************************A_InitCompensationDatas************************************************)
A_InitCompensationData();
(*********************************************************************btn_BCMove*****************************************************************)
IF InitPowerDone AND InitCompensationDatasDone THEN
	IF btn_BCGapMove THEN
		CASE m_state OF
			0:
				FB_Move.Mode:=5;						(*1£ºgapÄ£Ê½£»2£ºµ¥ÁºÄ£Ê½£¬3£ºtaperÄ£Ê½£¬4:DebugÄ£Ê½£¬5£º²¹³¥GapÄ£Ê½*)
				FB_Move.CoupleState:=st_Couple;			(*ñîºÏ×´Ì¬ÊäÈë*)
				FB_Move.PowerState:=st_Power;			(*µçÔ´×´Ì¬ÊäÈë*)
				FB_Move.BCGapMove:=TRUE;				(*Execute TRUE*)
				FB_Move.BCLeftTopPosition:=LeftTopLinPositionNew;(*Ã¿ÖáËÙ¶ÈÎ»ÖÃÊäÈë*)
				FB_Move.BCLeftTopVelocity:=BCGapVelocityNew/2;
				FB_Move.BCRightTopPosition:=RightTopLinPositionNew;
				FB_Move.BCRightTopVelocity:=BCGapVelocityNew/2;
				FB_Move.BCLeftBottomPosition:=LeftBottomLinPositionNew;
				FB_Move.BCLeftBottomVelocity:=BCGapVelocityNew/2;
				FB_Move.BCRightBottomPosition:=RightBottomLinPositionNew;
				FB_Move.BCRightBottomVelocity:=BCGapVelocityNew/2;
				FB_Move();								(*Æô¶¯FB*)
				IF LeftTopLinPositionNew-Pos_LeftTopLin>0.001 THEN	(*ÔË¶¯·½ÏòÖ¸Ê¾*)
					LeftTopLinMoveIndicator:=1;
				ELSIF LeftTopLinPositionNew-Pos_LeftTopLin<0.001 THEN
					LeftTopLinMoveIndicator:=-1;
				ELSE
					LeftTopLinMoveIndicator:=0;
				END_IF
				IF RightTopLinPositionNew-Pos_RightTopLin>0.001 THEN	(*ÔË¶¯·½ÏòÖ¸Ê¾*)
					RightTopLinMoveIndicator:=1;
				ELSIF RightTopLinPositionNew-Pos_RightTopLin<0.001 THEN
					RightTopLinMoveIndicator:=-1;
				ELSE
					RightTopLinMoveIndicator:=0;
				END_IF
				IF LeftBottomLinPositionNew-Pos_LeftBottomLin>0.001 THEN	(*ÔË¶¯·½ÏòÖ¸Ê¾*)
					LeftBottomLinMoveIndicator:=1;
				ELSIF LeftBottomLinPositionNew-Pos_LeftBottomLin<0.001 THEN
					LeftBottomLinMoveIndicator:=-1;
				ELSE
					LeftBottomLinMoveIndicator:=0;
				END_IF
				IF RightBottomLinPositionNew-Pos_RightBottomLin>0.001 THEN	(*ÔË¶¯·½ÏòÖ¸Ê¾*)
					RightBottomLinMoveIndicator:=1;
				ELSIF RightBottomLinPositionNew-Pos_RightBottomLin<0.001 THEN
					RightBottomLinMoveIndicator:=-1;
				ELSE
					RightBottomLinMoveIndicator:=0;
				END_IF
				m_state:=1;
			1:
				FB_Move();
				IF NOT FB_Move.BCGapDone THEN			(*ÔË¶¯Î´Íê³É£¬Ñ­»·*)
					Led_Run:=TRUE;
					m_state:=1;

				ELSE									(*ÔË¶¯Íê³É£¬ÏÂÒ»²½*)
					m_state:=88;
				END_IF
			88:
				btn_BCGapMove:=FALSE;					(*×´Ì¬»Ö¸´*)
				Led_Run:=FALSE;
				m_state:=0;
				LeftTopLinMoveIndicator:=0;
				RightTopLinMoveIndicator:=0;
				LeftBottomLinMoveIndicator:=0;
				RightBottomLinMoveIndicator:=0;
		END_CASE
	END_IF
END_IF
(*******************************************************************btn_Stop********************************************************************)
IF btn_BCGapStop THEN
	Led_Run:=FALSE;
	LeftTopLinMoveIndicator:=0;
	RightTopLinMoveIndicator:=0;
	LeftBottomLinMoveIndicator:=0;
	RightBottomLinMoveIndicator:=0;
	FB_Move.BCGapReset:=TRUE;							(*¸øÔË¶¯FB¸øÍ£Ö¹ÐÅºÅ£¬Ê¹FB_Move×´Ì¬»Ö¸´*)
	FB_Move();											(*Æô¶¯FB_Move*)
	btn_BCGapMove:=FALSE;								(*btn_GapMove:=FALSE*)
	m_state:=0;											(*m_state:=0;*)
	CASE s_state OF
			0:
				FB_Stop.Mode:=5;							(*1£ºgapÄ£Ê½£»2£ºµ¥ÁºÄ£Ê½£»3£ºtaperÄ£Ê½£»4£ºDebugÄ£Ê½£»5£ºBCGapÄ£Ê½*)
				FB_Stop.CoupleState:=st_Couple;			(*ñîºÏ×´Ì¬ÊäÈë*)
				FB_Stop.PowerState:=st_Power;				(*µçÔ´×´Ì¬ÊäÈë*)
				FB_Stop.BCGapStop:=TRUE;				(*Execute TRUE*)
				FB_Stop();								(*Æô¶¯FB*)
				s_state:=1;
			1:
				FB_Stop();
				IF NOT FB_Stop.BCGapDone THEN			(*Í£Ö¹Î´Íê³É£¬Ñ­»·*)
					s_state:=1;
				ELSE									(*Í£Ö¹Íê³É£¬ÏÂÒ»²½*)
					s_state:=88;
				END_IF
			88:
				btn_BCGapStop:=FALSE;						(*»Ö¸´×´Ì¬*)
				FB_Move.BCGapReset:=FALSE;				(*ÔËÐÐFB*)
				s_state:=0;
		END_CASE
END_IF
(*********************************************************************btn_PowerOff************************************************************)
IF btn_PowerOff THEN
	A_PowerOff();
END_IF
(*********************************************************************ÏÞÎ»Åö´¥×´Ì¬»Ö¸´************************************************************)
(*Èç¹û¼ì²âµ½ÏØÏÞÎ»¿ª¹ØÏÂ½µÑØ£¬»Ö¸´Move×´Ì¬*)
FTrig_ReachLS(CLK:=Unreach_LS_Top AND Unreach_LS_Bottom);
IF FTrig_ReachLS.Q THEN
	btn_BCGapStop:=TRUE;
END_IF
(*Èç¹û¼ì²âµ½TopÏÞÎ»¿ª¹ØFALSE£¬ÇÒÄ¿±êÎ»ÖÃ´óÓÚµ±Ç°Î»ÖÃÊ±£¬»òÕßÏà·´Ê±£¬»Ö¸´Move×´Ì¬*)
IF NOT Unreach_LS_Top AND BCGapPositionNew-BCGapPositionDisplay>0.0005 AND btn_BCGapMove THEN
	btn_BCGapStop:=TRUE;
END_IF
IF NOT Unreach_LS_Bottom AND BCGapPositionNew-BCGapPositionDisplay<0.0005 AND btn_BCGapMove THEN
	btn_BCGapStop:=TRUE;
END_IF

ACTION A_InitCompensationData:
(*BCGapPositionNewºÍBCGapVelocityNew³¬³ö·¶Î§£¬ESTOP*)
(*IF BCGapPositionNew<-100 OR BCGapPositionNew>400 THEN
	btn_BCGapStop:=TRUE;
	FB_PlcEmergencyStop();
	Error:=TRUE;
	ErrorID:=20;
	LED_Error:=TRUE;
	InitCompensationDatasDone:=FALSE;
ELSIF  BCGapVelocityNew<0 OR  BCGapVelocityNew>2 THEN
	btn_BCGapStop:=TRUE;
	FB_PlcEmergencyStop();
	Error:=TRUE;
	ErrorID:=21;
	LED_Error:=TRUE;
	InitCompensationDatasDone:=FALSE;
END_IF
*)
(*¸ù¾ÝÊäÈëGapPosition²¹³¥²¢·Ö½âµ½Ã¿¸öÖá£¬¼ÆËãÃ¿¸öÖáµÄÎ»ÖÃ*)
IF USE_SingleAxis_Compensation THEN
	(*IF LeftTopLin.Status.NotMoving AND RightTopLin.Status.NotMoving AND LeftBottomLin.Status.NotMoving AND RightBottomLin.Status.NotMoving THEN*)
		FOR	i:= 1 TO 17 DO
			IF BCGapPositionNew/2<M_Compensation[i+1].Encoder AND BCGapPositionNew/2>=M_Compensation[i].Encoder THEN
				IF i<>18 THEN
					LeftTopLinPositionNew:=(((BCGapPositionNew/2-M_Compensation[i].Encoder)*(M_Compensation[i+1].LeftTop-M_Compensation[i].LeftTop))
							/(M_Compensation[i+1].Encoder-M_Compensation[i].Encoder))+M_Compensation[i].LeftTop;
					RightTopLinPositionNew:=(((BCGapPositionNew/2-M_Compensation[i].Encoder)*(M_Compensation[i+1].RightTop-M_Compensation[i].RightTop))
							/(M_Compensation[i+1].Encoder-M_Compensation[i].Encoder))+M_Compensation[i].RightTop;
					LeftBottomLinPositionNew:=(((BCGapPositionNew/2-M_Compensation[i].Encoder)*(M_Compensation[i+1].LeftBottom-M_Compensation[i].LeftBottom))
							/(M_Compensation[i+1].Encoder-M_Compensation[i].Encoder))+M_Compensation[i].LeftBottom;
					RightBottomLinPositionNew:=(((BCGapPositionNew/2-M_Compensation[i].Encoder)*(M_Compensation[i+1].RightBottom-M_Compensation[i].RightBottom))
							/(M_Compensation[i+1].Encoder-M_Compensation[i].Encoder))+M_Compensation[i].RightBottom;
					M_CompensationNumber:=i;
					InitCompensationDatasDone:=TRUE;
(*
					(*¸ù¾ÝÃ¿¸öÖáµÄÊµ¼ÊÎ»ÖÃ£¬·´ËãÐèÒªÔÚ¿ØÖÆÏµÍ³UIÖÐÏÔÊ¾µÄÎ»ÖÃ*)
					LeftTopLinPositionDisplay:=(((M_Compensation[i+1].Encoder-M_Compensation[i].Encoder)*(Pos_LeftTopLin-M_Compensation[i].LeftTop))
							/(M_Compensation[i+1].LeftTop-M_Compensation[i].LeftTop))+M_Compensation[i].Encoder;
					RightTopLinPositionDisplay:=(((M_Compensation[i+1].Encoder-M_Compensation[i].Encoder)*(Pos_RightTopLin-M_Compensation[i].RightTop))
							/(M_Compensation[i+1].RightTop-M_Compensation[i].LeftTop))+M_Compensation[i].Encoder;
					LeftBottomLinPositionDisplay:=(((M_Compensation[i+1].Encoder-M_Compensation[i].Encoder)*(Pos_LeftBottomLin-M_Compensation[i].LeftBottom))
							/(M_Compensation[i+1].LeftBottom-M_Compensation[i].LeftBottom))+M_Compensation[i].Encoder;
					RightBottomLinPositionDisplay:=(((M_Compensation[i+1].Encoder-M_Compensation[i].Encoder)*(Pos_RightBottomLin-M_Compensation[i].RightBottom))
							/(M_Compensation[i+1].RightBottom-M_Compensation[i].RightBottom))+M_Compensation[i].Encoder;
*)
				ELSIF i=18 AND BCGapPositionNew/2=M_Compensation[i].Encoder THEN		(*Gap=14µÄÌØÊâÇé¿ö*)
					(**)
					LeftTopLinPositionNew:=M_Compensation[i].LeftTop;
					RightTopLinPositionNew:=M_Compensation[i].RightTop;
					LeftBottomLinPositionNew:=M_Compensation[i].LeftBottom;
					RightBottomLinPositionNew:=M_Compensation[i].RightBottom;
					(*
					LeftTopLinPositionDisplay:=(((M_Compensation[i+1].Encoder-M_Compensation[i].Encoder)*(Pos_LeftTopLin-M_Compensation[i].LeftTop))
							/(M_Compensation[i+1].LeftTop-M_Compensation[i].LeftTop))+M_Compensation[i].Encoder;
					RightTopLinPositionDisplay:=(((M_Compensation[i+1].Encoder-M_Compensation[i].Encoder)*(Pos_RightTopLin-M_Compensation[i].RightTop))
							/(M_Compensation[i+1].RightTop-M_Compensation[i].LeftTop))+M_Compensation[i].Encoder;
					LeftBottomLinPositionDisplay:=(((M_Compensation[i+1].Encoder-M_Compensation[i].Encoder)*(Pos_LeftBottomLin-M_Compensation[i].LeftBottom))
							/(M_Compensation[i+1].LeftBottom-M_Compensation[i].LeftBottom))+M_Compensation[i].Encoder;
					RightBottomLinPositionDisplay:=(((M_Compensation[i+1].Encoder-M_Compensation[i].Encoder)*(Pos_RightBottomLin-M_Compensation[i].RightBottom))
							/(M_Compensation[i+1].RightBottom-M_Compensation[i].RightBottom))+M_Compensation[i].Encoder;
*)
					M_CompensationNumber:=i;
					InitCompensationDatasDone:=TRUE;
				ELSE(*Gap>14µÄÇé¿ö*)
					LeftTopLinPositionNew:=BCGapPositionNew/2;
					RightTopLinPositionNew:=BCGapPositionNew/2;
					LeftBottomLinPositionNew:=BCGapPositionNew/2;
					RightBottomLinPositionNew:=BCGapPositionNew/2;
					(*
					LeftTopLinPositionDisplay:=Pos_LeftTopLin;
					RightTopLinPositionDisplay:=Pos_RightTopLin;
					LeftBottomLinPositionDisplay:=Pos_LeftBottomLin;
					RightBottomLinPositionDisplay:=Pos_RightBottomLin;
*)
					M_CompensationNumber:=i;
					InitCompensationDatasDone:=TRUE;
				END_IF
			END_IF
		END_FOR

		FOR j:= 1 TO 17 DO
			IF Pos_RightBottomLin<M_Compensation[j+1].RightBottom AND Pos_RightBottomLin>=M_Compensation[j].RightBottom THEN
				IF j<>18 THEN
					(*¸ù¾ÝÃ¿¸öÖáµÄÊµ¼ÊÎ»ÖÃ£¬·´ËãÐèÒªÔÚ¿ØÖÆÏµÍ³UIÖÐÏÔÊ¾µÄÎ»ÖÃ*)
					LeftTopLinPositionDisplay:=(((M_Compensation[j+1].Encoder-M_Compensation[j].Encoder)*(Pos_LeftTopLin-M_Compensation[j].LeftTop))
							/(M_Compensation[j+1].LeftTop-M_Compensation[j].LeftTop))+M_Compensation[j].Encoder;
					RightTopLinPositionDisplay:=(((M_Compensation[j+1].Encoder-M_Compensation[j].Encoder)*(Pos_RightTopLin-M_Compensation[j].RightTop))
							/(M_Compensation[j+1].RightTop-M_Compensation[j].RightTop))+M_Compensation[j].Encoder;
					LeftBottomLinPositionDisplay:=(((M_Compensation[j+1].Encoder-M_Compensation[j].Encoder)*(Pos_LeftBottomLin-M_Compensation[j].LeftBottom))
							/(M_Compensation[j+1].LeftBottom-M_Compensation[j].LeftBottom))+M_Compensation[j].Encoder;
					RightBottomLinPositionDisplay:=(((M_Compensation[j+1].Encoder-M_Compensation[j].Encoder)*(Pos_RightBottomLin-M_Compensation[j].RightBottom))
							/(M_Compensation[j+1].RightBottom-M_Compensation[j].RightBottom))+M_Compensation[j].Encoder;
					M_DisplayNumber:=j;
				ELSIF j=18 AND BCGapPositionNew/2=M_Compensation[j].Encoder THEN		(*Gap=14µÄÌØÊâÇé¿ö*)
					(**)
					LeftTopLinPositionDisplay:=(((M_Compensation[j+1].Encoder-M_Compensation[j].Encoder)*(Pos_LeftTopLin-M_Compensation[j].LeftTop))
							/(M_Compensation[j+1].LeftTop-M_Compensation[j].LeftTop))+M_Compensation[j].Encoder;
					RightTopLinPositionDisplay:=(((M_Compensation[j+1].Encoder-M_Compensation[j].Encoder)*(Pos_RightTopLin-M_Compensation[j].RightTop))
							/(M_Compensation[j+1].RightTop-M_Compensation[j].LeftTop))+M_Compensation[j].Encoder;
					LeftBottomLinPositionDisplay:=(((M_Compensation[j+1].Encoder-M_Compensation[j].Encoder)*(Pos_LeftBottomLin-M_Compensation[j].LeftBottom))
							/(M_Compensation[j+1].LeftBottom-M_Compensation[j].LeftBottom))+M_Compensation[j].Encoder;
					RightBottomLinPositionDisplay:=(((M_Compensation[j+1].Encoder-M_Compensation[j].Encoder)*(Pos_RightBottomLin-M_Compensation[j].RightBottom))
							/(M_Compensation[j+1].RightBottom-M_Compensation[j].RightBottom))+M_Compensation[j].Encoder;
					M_DisplayNumber:=j;
				ELSE(*Gap>14µÄÇé¿ö*)
					(**)
					LeftTopLinPositionDisplay:=Pos_LeftTopLin;
					RightTopLinPositionDisplay:=Pos_RightTopLin;
					LeftBottomLinPositionDisplay:=Pos_LeftBottomLin;
					RightBottomLinPositionDisplay:=Pos_RightBottomLin;
					M_DisplayNumber:=j;
				END_IF
			END_IF
		END_FOR
	(*END_IF*)
ELSE
	LeftTopLinPositionNew:=BCGapPositionNew/2;
	RightTopLinPositionNew:=BCGapPositionNew/2;
	LeftBottomLinPositionNew:=BCGapPositionNew/2;
	RightBottomLinPositionNew:=BCGapPositionNew/2;
	LeftTopLinPositionDisplay:=Pos_LeftTopLin;
	RightTopLinPositionDisplay:=Pos_RightTopLin;
	LeftBottomLinPositionDisplay:=Pos_LeftBottomLin;
	RightBottomLinPositionDisplay:=Pos_RightBottomLin;
	M_CompensationNumber:=0;
	InitCompensationDatasDone:=TRUE;
END_IF

LeftTopLinVelocityDisplay:=Velo_LeftTopLin;
RightTopLinVelocityDisplay:=Velo_RightTopLin;
LeftBottomLinVelocityDisplay:=Velo_LeftBottomLin;
RightBottomLinVelocityDisplay:=Velo_RightBottomLin;
END_ACTION

ACTION A_MonitoringAllAxis:
(****************************************************************
NAME:			A_MonitoringAllAxis
DATA:			2018.1.9
VERSION:		1.0.0
DESCRIPTION:	
				Ã¿´ÎÑ­»·¾ùÖ´ÐÐÖáÎ»ÖÃºÍÖáÔË¶¯µÄ¼ì²é
				2.4Öá¹âÕ¤³ßÎ»ÖÃ¡¢ËÙ¶È¶Ô±È¼ì²é
HISTORY:
				2017.1.9		NEW

***************************************************************)

(*************************************************************************************2.4Öá¹âÕ¤³ßÎ»ÖÃ¡¢ËÙ¶È¶Ô±È¼ì²é**********************************************************************)
IF  st_Power<>0 THEN
CASE moni_State OF
(*Top Î»ÖÃºÍËÙ¶È±È¶Ô*)
0:
		(*Î»ÖÃ*)
		(*Top*)
		Diff_BCTopPos_actual:=ABS(Pos_leftTopLin-Pos_RightTopLin);
		(*Bottom*)
		Diff_BCBottomPos_actual:=ABS(Pos_LeftBottomLin-Pos_RightBottomLin);
		(*Left*)
		Diff_BCLeftPos_actual:=ABS(Pos_LeftTopLin-Pos_LeftBottomLin);
		(*Right*)
		Diff_BCRightPos_actual:=ABS(Pos_RightTopLin-Pos_RightBottomLin);
		(*ËÙ¶È*)
		(*Top*)
		Diff_BCTopVelo_actual:=ABS(Velo_leftTopLin-Velo_RightTopLin);
		(*Bottom*)
		Diff_BCBottomVelo_actual:=ABS(Velo_LeftBottomLin-Velo_RightBottomLin);
		(*Left*)
		Diff_BCLeftVelo_actual:=ABS(Velo_LeftTopLin-Velo_LeftBottomLin);
		(*Right*)
		Diff_BCRightVelo_actual:=ABS(Velo_RightTopLin-Velo_RightBottomLin);
		IF Diff_BCTopPos_actual >Threshold_BCTopPos THEN
				ErrorID:=11;
				moni_State:=-100;
		ELSIF Diff_BCTopVelo_actual>Threshold_BCTopVelo  THEN
				ErrorID:=12;
				moni_State:=-100;
		(*Bottom Î»ÖÃºÍËÙ¶È±È¶Ô*)
		ELSIF Diff_BCBottomPos_actual>Threshold_BCBottomPos THEN
				ErrorID:=13;
				moni_State:=-100;
		ELSIF Diff_BCBottomVelo_actual>Threshold_BCBottomVelo  THEN
				ErrorID:=14;
				moni_State:=-100;
		(*Left Î»ÖÃºÍËÙ¶È±È¶Ô*)
		ELSIF Diff_BCLeftPos_actual>Threshold_BCLeftPos  THEN
				ErrorID:=15;
				moni_State:=-100;
		ELSIF  Diff_BCLeftVelo_actual>Threshold_BCLeftVelo THEN
				ErrorID:=16;
				moni_State:=-100;
		(*Right Î»ÖÃºÍËÙ¶È±È¶Ô*)
		ELSIF Diff_BCRightPos_actual>Threshold_BCRightPos  THEN
				ErrorID:=17;
				moni_State:=-100;
		ELSIF  Diff_BCRightVelo_actual>Threshold_BCRightVelo THEN
				ErrorID:=18;
				moni_State:=-100;
		END_IF
-100:
		btn_BCGapStop:=TRUE;
		FB_PlcEmergencyStop();
		Error:=TRUE;
		LED_Error:=TRUE;
END_CASE
END_IF
END_ACTION

ACTION A_PosDiffDetection:
IF ABS(PosDiff_LeftTopLin_actual-PosDiff_RightTopLin_actual)>0.2 THEN		(*ÉÏÖá×óÓÒLagDistanceÖ®²î*)
	ErrorID:=51;
	Error:=TRUE;
	btn_BCGapStop:=TRUE;
	FB_PlcEmergencyStop();
	LED_Error:=TRUE;
ELSIF ABS(PosDiff_LeftBottomLin_actual-PosDiff_RightBottomLin_actual)>0.2 THEN
	ErrorID:=53;
	Error:=TRUE;
	btn_BCGapStop:=TRUE;
	FB_PlcEmergencyStop();
	LED_Error:=TRUE;
END_IF
END_ACTION

ACTION A_PowerOff:
CASE d_state OF
		0:(*PowerOff*)
			FB_Power(Off:=TRUE);
				d_state:=1;
		1:
			IF NOT FB_power.OffStatus THEN
				d_state:=1;
			ELSE
				d_state:=88;
			END_IF
		88:(*ResetAllState*)
			btn_PowerOn:=FALSE;
			btn_BCGapMove:=FALSE;
			btn_BCGapStop:=FALSE;
			LeftTopLinMoveIndicator:=0;
			RightTopLinMoveIndicator:=0;
			LeftBottomLinMoveIndicator:=0;
			RightBottomLinMoveIndicator:=0;
			fb_ton1.IN:=FALSE;
			fb_ton2.IN:=FALSE;
			fb_ton3.IN:=FALSE;
			State:=0;
			Busy:=FALSE;
			InitPowerDone:=FALSE;
			InitCompensationDatasDone:=FALSE;
			Error:=FALSE;
			ErrorID:=0;
			m_state:=0;
			s_state:=0;
			btn_PowerOff:=FALSE;
			d_state:=0;
			Led_Run:=FALSE;
			Led_Error:=FALSE;
			moni_State:=0;
			i:=0;
END_CASE
END_ACTION

ACTION A_PowerOn:
(****************************************************************
NAME:			A_PowerOn
DATA:			2018.1.9
VERSION:		1.0.0
DESCRIPTION:	
				ÉÏµãÃüÁîºó£¬Ë³ÐòÖ´ÐÐ£º
				1.FB_PowerOn
				·µ»ØÖ´ÐÐÊÇ·ñ³É¹¦
HISTORY:
				2019.1.9		NEW

***************************************************************)
fb_ton3(PT:=t#0.5s);
CASE State OF
	0:	(*FB_Power_On*)
		FB_Power(On:=TRUE);
		fb_ton3.IN:=TRUE;
		State:=1;
	1:	(*wait*)
		FB_power();
		IF NOT FB_power.OnStatus THEN		(*FB_Power_OnÃ»ÓÐÖ´ÐÐÍê£¬wait£¬³¬Ê±FB Error*)
			IF NOT fb_ton3.Q THEN
				State:=1;
			ELSE
				ErrorID:=1;
				State:=99;
			END_IF
		ELSE
			State:=88;
		END_IF
	88:	(*All Done*)
		btn_PowerOn:=FALSE;
		State:=0;
		Error:=FALSE;
		ErrorID:=0;
		Busy:=FALSE;
		InitPowerDone:=TRUE;
		FB_power.On:=FALSE;
		fb_ton3.IN:=FALSE;
		LED_Error:=FALSE;
	99:
		btn_PowerOn:=FALSE;
		State:=99;
		Error:=TRUE;
		Busy:=FALSE;
		InitPowerDone:=FALSE;
		fb_ton3.IN:=FALSE;
		LED_Error:=TRUE;
END_CASE
END_ACTION

END_PROGRAM

// ---- POUs/0.UserMode/UserMode.TcPOU
PROGRAM UserMode
VAR
(*key Command*)
	btn_Power:BOOL;
	btn_PowerOn: BOOL;
	btn_PowerOff: BOOL;
(*GapMode*)
	UserGapPositionNew:LREAL:=20;//target
	UserGapVelocityNew:LREAL:=1;//target
	UserGapPositionDisplay:LREAL;//current
	UserGapVelocityDisplay:LREAL;//current
	UserTaperPositionNew:LREAL:=0;//target
	UserTaperVelocityNew:LREAL:=1;//target
	UserTaperPositionDisplay:LREAL;//current
	//UserTaperPositionDisplay_FromRightTop:LREAL;
	//UserTaperPositionDisplay_FromRightBottom:LREAL;
	UserTaperVelocityDisplay:LREAL;//target
	//Pos_LeftTopLin_NoTaper:LREAL;
	//Pos_RightTopLin_NoTaper:LREAL;
	//Pos_LeftBottomLin_NoTaper:LREAL;
	//Pos_RightBottomLin_NoTaper:LREAL;
	UserGapPositionDisplay_FromLeftTop:LREAL;
	UserGapPositionDisplay_FromLeftBottom:LREAL;
	//
	UserRightGapPositionNew:LREAL;
	UserRightGapVelocityNew:LREAL;
	UserRightGapPositionDisplay:LREAL;
	UserRightGapVelocityDisplay:LREAL;
	UserRightGapPositionDisplay_FromRightTop:LREAL;
	UserRightGapPositionDisplay_FromRightBottom:LREAL;
	(**)
	btn_UserGapMove:BOOL;
	btn_UserGapStop:BOOL;
	(*Var*)
	fb_ton1:TON;
	fb_ton2:TON;
	fb_ton3:TON;
	(*Status*)
	State:DINT;
	Busy:BOOL;
	InitPowerDone:BOOL;
	InitCompensationDatasDone:BOOL;
	(*FB*)
	m_state: DINT;
	n_state: DINT;
	s_state: DINT;
	(*¼ì²âµ½ÏÞÎ»£¬»Ö¸´Move×´Ì¬*)
	FTrig_ReachLS: F_TRIG;
	FTrig_btn_GapMove: F_TRIG;
	GapOutRange: BOOL;
	(*PowerOff*)
	d_state: DINT;
	i: INT;
	j: INT;
	k: INT;
	moni_State:DINT;
	TargetPosLessThanCurrentPos:BOOL;
	TargetLTPosLessThanCurrentLTPos:BOOL;
	TargetRTPosLessThanCurrentRTPos:BOOL;
	TargetLBPosLessThanCurrentLBPos:BOOL;
	TargetRBPosLessThanCurrentRBPos:BOOL;
	PositiveMoving:BOOL;
	HysteresisMoving:BOOL;
	NoneHysteresisMoving:BOOL;
	(*Spectroscopy scanning Mode*)
	IsSSMotionMode:BOOL;
	RegularMotionMode:BOOL;
	SSMotionMode:BOOL;
	SS_StepSize:LREAL:=0.001;
	SS_StepNumber:INT:=10;
	SS_StepVelocity:LREAL:=1;
	SS_Move:BOOL;
	SS_Stop:BOOL;
	SS_MoveState:DINT;
	SS_StopState:DINT;
	SS_currentStep:DINT:=0;
	SS_StepSystemTime_Begin:ARRAY[0..100] OF ULINT;
	SS_StepSystemTime_End:ARRAY[0..100] OF ULINT;
	SS_StepCountTime:ARRAY[0..100] OF ULINT;
	SS_TimeCountBegin:BOOL;
	m: INT;
	SS_TON: TON;
	StepEachTime:TIME;
	StepEachTime_ms:INT:=1000;//ms
	SS_OTSTRUCT :OTSTRUCT ;
	SS_StartPositionDisplay:LREAL;
	RTRG_SS_StartPositionDisplay:R_TRIG;
	SS_InitStartPositionDone:BOOL;
	(*input protection*)
	//
	min_UserGapPositionNew:LREAL:=10;
	max_UserGapPositionNew:LREAL:=200;
	inRange_UserGapPositionNew:BOOL;
	//
	min_UserGapVelocityNew:LREAL:=0;
	max_UserGapVelocityNew:LREAL:=3;
	inRange_UserGapVelocityNew:BOOL;
	//
	min_UserTaperPositionNew: LREAL:=0;;
	max_UserTaperPositionNew: LREAL:=4;
	inRange_UserTaperPositionNew: BOOL;
	//
	min_UserTaperVelocityNew: LREAL:=0;
	max_UserTaperVelocityNew: LREAL:=1;
	inRange_UserTaperVelocityNew: BOOL;
	//
	min_SS_StepSize	: LREAL:=0;
	max_SS_StepSize	: LREAL:=200;
	inRange_SS_StepSize	: BOOL;
	//
	min_SS_StepNumber	: INT:=1;
	max_SS_StepNumber	: INT:=1000;
	inRange_SS_StepNumber	: BOOL;
	//
	min_SS_StepVelocity:LREAL:=0;
	max_SS_StepVelocity:LREAL:=1;
	inRange_SS_StepVelocity:BOOL;
	//
	min_StepEachTime_ms:INT:=100;
	max_StepEachTime_ms:INT:=10000;
	inRange_StepEachTime_ms:BOOL;
	l: INT;
	Threshold_UserTopPos_PLC: LREAL;
	Threshold_UserTopVelo_PLC: LREAL;
	Threshold_UserBottomPos_PLC: LREAL;
	Threshold_UserBottomVelo_PLC: LREAL;
	Threshold_UserLeftPos_PLC: LREAL;
	Threshold_UserLeftVelo_PLC: LREAL;
	Threshold_UserRightPos_PLC: LREAL;
	Threshold_UserRightVelo_PLC: LREAL;
	testa: BOOL;
	testb: BOOL;
	Threshold_GapChangeFlag: LREAL;
	Threshold_TaperChangeFlag: LREAL;
	TaperAndGapSafetyfactor: LREAL:=1;
END_VAR

IF NOT PositionBiasDone THEN
	RETURN;
END_IF
IF NOT loadParametersDone THEN
	RETURN;
END_IF
(*btn_Power On/Off*)
IF btn_Power AND NOT st_Power THEN
	btn_PowerOn:=TRUE;
	btn_Power:=FALSE;
END_IF
IF btn_Power AND st_Power THEN
	btn_PowerOff:=TRUE;
	btn_Power:=FALSE;
END_IF
IF btn_PowerOn THEN
	A_PowerOn();
END_IF
IF btn_PowerOff THEN
	A_PowerOff();
END_IF

(*检查couple状态，不允许couple*)
A_CheckCoupleStatus();

(*监控四轴位置速度等*)
A_MonitoringAllAxis();

(*补偿数据处理*)
A_InitCompensationData();

(*常规磁间隙开合*)
IF RegularMotionMode AND NOT SSMotionMode THEN
	A_RegularMotion();
END_IF

